(* CoDeSys 2.3.9.47 project: 3floor_2016_11_08_spalnya_fancoil_speed_temporary_change.prx *)
(* Libraries: TcEIB.lbx 16.5.14 13:12:22, TcSystemBX.lbx 11.6.12 12:56:16, TcBABasicBX.lbx 22.7.15 14:46:56, TcBaseBX.lbx 10.5.06 07:50:20, standard.lbx 5.12.03 07:02:30 *)

(* Task configuration *)
TASK Standard (PRIORITY := 0, INTERVAL := T#20ms);
	MAIN
END_TASK

(* Global variable list: M_Var_1 *)
VAR_GLOBAL
	data1floor: ARRAY[0..200] OF BYTE;
	data1floor_prev: ARRAY[0..200] OF BYTE;
	ads_adr1: STRING:='10.0.5.61.1.1';

	fb_komora_l_send_status_ex: 			EIB_BIT_SEND_EX;
	fb_su1_l_send_status_ex: 				EIB_BIT_SEND_EX;
	fb_topochna_l_send_status_ex: 			EIB_BIT_SEND_EX;
	fb_su2_bra_send_status_ex: 				EIB_BIT_SEND_EX;
	fb_topochna2_l_send_status_ex: 		EIB_BIT_SEND_EX;
	fb_su2_l_send_status_ex: 				EIB_BIT_SEND_EX;
	fb_su1_rakovyna_send_status_ex: 		EIB_BIT_SEND_EX;
	fb_su2_dush_send_status_ex: 			EIB_BIT_SEND_EX;
	fb_dush_send_status_ex: 				EIB_BIT_SEND_EX;
	fb_vitalnya_smugy2_send_status_ex: 		EIB_BIT_SEND_EX;
	fb_su2_polytsi_send_status_ex: 			EIB_BIT_SEND_EX;
	fb_kuhnya1_send_status_ex: 			EIB_BIT_SEND_EX;
	fb_kuhnya2_send_status_ex: 			EIB_BIT_SEND_EX;
	fb_vitalnya_smugy1_send_status_ex: 		EIB_BIT_SEND_EX;
	fb_vitalnya_l_send_status_ex: 			EIB_BIT_SEND_EX;
	fb_vitalnya_prokladka_send_status_ex: 	EIB_BIT_SEND_EX;
	fb_terassa_stina_send_status_ex: 		EIB_BIT_SEND_EX;
	fb_pidval_shody_send_status_ex: 		EIB_BIT_SEND_EX;
	fb_skhody2pov_send_status_ex: 			EIB_BIT_SEND_EX;
	fb_tambur_l_send_status_ex: 			EIB_BIT_SEND_EX;
	fb_vent_su1_send_status_ex: 			EIB_BIT_SEND_EX;
	fb_vent_kuh_low_send_status_ex: 		EIB_BIT_SEND_EX;
	fb_vent_dush_send_status_ex: 			EIB_BIT_SEND_EX;
	fb_vent_komora_send_status_ex: 		EIB_BIT_SEND_EX;
	fb_vent_kuh_high_send_status_ex: 		EIB_BIT_SEND_EX;
	fb_floor1_lights_send_status_ex: 			EIB_BIT_SEND_EX;

	fb_komora_l_read: 			EIB_BIT_REC;
	fb_su1_l_read: 				EIB_BIT_REC;
	fb_topochna_l_read: 		EIB_BIT_REC;
	fb_su2_bra_read: 			EIB_BIT_REC;
	fb_topochna2_l_read: 		EIB_BIT_REC;
	fb_su2_l_read: 				EIB_BIT_REC;
	fb_su1_rakovyna_read: 		EIB_BIT_REC;
	fb_su2_dush_read: 			EIB_BIT_REC;
	fb_dush_read: 				EIB_BIT_REC;
	fb_vitalnya_smugy2_read: 	EIB_BIT_REC;
	fb_su2_polytsi_read: 		EIB_BIT_REC;
	fb_kuhnya1_read: 			EIB_BIT_REC;
	fb_kuhnya2_read: 			EIB_BIT_REC;
	fb_vitalnya_smugy1_read: 	EIB_BIT_REC;
	fb_vitalnya_l_read: 			EIB_BIT_REC;
	fb_vitalnya_prokladka_read: 	EIB_BIT_REC;
	fb_terassa_stina_read: 		EIB_BIT_REC;
	fb_pidval_shody_read: 		EIB_BIT_REC;
	fb_skhody2pov_read: 		EIB_BIT_REC;
	fb_tambur_l_read: 			EIB_BIT_REC;
	fb_vent_su1_read: 			EIB_BIT_REC;
	fb_vent_kuh_low_read: 		EIB_BIT_REC;
	fb_vent_dush_read: 			EIB_BIT_REC;
	fb_vent_komora_read: 		EIB_BIT_REC;
	fb_vent_kuh_high_read: 		EIB_BIT_REC;
	fb_floor1_lights_read: 		EIB_BIT_REC;

	moove_garderob				AT%MX100.0:BOOL;
	moove_tambur					AT%MX100.1:BOOL;
	moove_dytjacha					AT%MX100.2:BOOL;
	moove_spalnya					AT%MX100.3:BOOL;
	moove_korydor					AT%MX100.4:BOOL;
	moove_skhody					AT%MX100.5:BOOL;

	komora_l 						AT%MX101.0:BOOL;
	su1_l 							AT%MX101.1:BOOL;
	topochna_l 						AT%MX101.2:BOOL;
	su2_bra	 						AT%MX101.3:BOOL;
	su2_l 							AT%MX101.4:BOOL;
	su1_rakovyna 					AT%MX101.5:BOOL;
	su2_dush 						AT%MX101.6:BOOL;
	dush 							AT%MX101.7:BOOL;

	kuhnya1	 					AT%MX102.0:BOOL;
	vitalnya_smugy1 				AT%MX102.1:BOOL;
	vitalnya_l 						AT%MX102.2:BOOL;
	vitalnya_prokladka 				AT%MX102.3:BOOL;
	terassa_stina	 				AT%MX102.4:BOOL;
	pidval_shody	 				AT%MX102.5:BOOL;
	skhody2pov 					AT%MX102.6:BOOL;
	tambur_l 						AT%MX102.7:BOOL;

	vent_su1 						AT%MX103.0:BOOL;
	vent_kuh_low 					AT%MX103.1:BOOL;
	vent_dush 						AT%MX103.2:BOOL;
	vent_komora 					AT%MX103.3:BOOL;
	vent_kuh_high 					AT%MX103.4:BOOL;

	floor1_lights:						BOOL;

END_VAR

(* Global variable list: M_Var_2 *)
VAR_GLOBAL
	data2floor: ARRAY[0..300] OF BYTE;
	data2floor_prev: ARRAY[0..300] OF BYTE;
	ads_adr2: STRING:='10.0.5.62.1.1';

	fb_balkon_peryla_send_status_ex: 			EIB_BIT_SEND_EX;
	fb_kino_l_send_status_ex:  					EIB_BIT_SEND_EX;
	fb_balkon_bra_send_status_ex: 				EIB_BIT_SEND_EX;
	fb_kabinet_balkon_l_send_status_ex:  		EIB_BIT_SEND_EX;
	fb_balkon_send_status_ex:					EIB_BIT_SEND_EX;
	fb_korydor1_send_status_ex:	 				EIB_BIT_SEND_EX;
	fb_kino_bra_send_status_ex:					EIB_BIT_SEND_EX;
	fb_kino_bra_send_dim_status_ex:			EIB_8BIT_SIGN_SEND_EX;
	fb_studio_pidsvitka_send_status_ex: 			EIB_BIT_SEND_EX;
	fb_skhody2_3_send_status_ex:	  			EIB_BIT_SEND_EX;
	fb_studio_l_send_status_ex:	 				EIB_BIT_SEND_EX;
	fb_kabinet_svitlo_send_status_ex:			EIB_BIT_SEND_EX;
	fb_stend_send_status_ex:  					EIB_BIT_SEND_EX;
	fb_kabinet_kobra_send_status_ex:  			EIB_BIT_SEND_EX;
	fb_skhody_peryla_send_status_ex:  			EIB_BIT_SEND_EX;
	fb_tambur2_send_status_ex: 					EIB_BIT_SEND_EX;
	fb_floor2_lights_send_status_ex: 				EIB_BIT_SEND_EX;

	fb_balkon_peryla_read: 						EIB_BIT_REC;
	fb_kino_l_read:  								EIB_BIT_REC;
	fb_balkon_bra_read: 						EIB_BIT_REC;
	fb_kabinet_balkon_l_read:  					EIB_BIT_REC;
	fb_balkon_read:								EIB_BIT_REC;
	fb_korydor1_read:							EIB_BIT_REC;
	fb_kino_bra_read:							EIB_BIT_REC;
	fb_kino_bra_dim_read:						EIB_8BIT_SIGN_REC;
	fb_studio_pidsvitka_read: 					EIB_BIT_REC;
	fb_skhody2_3_read:	  						EIB_BIT_REC;
	fb_studio_l_read:	 						EIB_BIT_REC;
	fb_kabinet_svitlo_read:						EIB_BIT_REC;
	fb_stend_read:  								EIB_BIT_REC;
	fb_kabinet_kobra_read:  						EIB_BIT_REC;
	fb_skhody_peryla_read:  						EIB_BIT_REC;
	fb_tambur2_read: 							EIB_BIT_REC;
	fb_floor2_lights_read: 						EIB_BIT_REC;


	eib_shtory_kino, eib_tul_kino: 				EIB_BIT_REC; (*ловлять в мережі смартбаса телеграмки для штор і тюлей*)
	eib_shtory_kabinet, eib_tul_kabinet: 			EIB_BIT_REC;

	fb_eib_shtory_kino_move:					EIB_BIT_REC;
	fb_eib_shtory_kino_position:					EIB_8BIT_SIGN_REC;
	fb_eib_shtory_kino_actualPosition:			EIB_8BIT_SIGN_SEND;

	fb_eib_tul_kino_move:						EIB_BIT_REC;
	fb_eib_tul_kino_position:						EIB_8BIT_SIGN_REC;
	fb_eib_tul_kino_actualPosition:				EIB_8BIT_SIGN_SEND;

	fb_eib_shtory_kabinet_move:					EIB_BIT_REC;
	fb_eib_shtory_kabinet_position:				EIB_8BIT_SIGN_REC;
	fb_eib_shtory_kabinet_actualPosition:			EIB_8BIT_SIGN_SEND;

	fb_eib_tul_kabinet_move:					EIB_BIT_REC;
	fb_eib_tul_kabinet_position:					EIB_8BIT_SIGN_REC;
	fb_eib_tul_kabinet_actualPosition:			EIB_8BIT_SIGN_SEND;






	balkon_peryla					AT%MX200.0:BOOL;
	kino_l							AT%MX200.1:BOOL;
	balkon_bra						AT%MX200.2:BOOL;
	kabinet_balkon_l				AT%MX200.3:BOOL;
	balkon							AT%MX200.4:BOOL;
	korydor1						AT%MX200.5:BOOL;
	kino_bra						AT%MX200.6:BOOL;
	studio_pidsvitka					AT%MX200.7:BOOL;

	skhody2_3						AT%MX201.0:BOOL;
	studio_l							AT%MX201.1:BOOL;
	kabinet_svitlo					AT%MX201.2:BOOL;
	kabinet_kobra					AT%MX201.3:BOOL;
	tambur2							AT%MX201.4:BOOL;
	stend							AT%MX201.5:BOOL;
	skhody_peryla					AT%MX201.6:BOOL;

	kino_bra_dim_value				AT%MB202:BYTE;

	collector_kabinet1					AT%MX203.0:BOOL;
	collector_kabinet2					AT%MX203.1:BOOL;
	collector_studio1					AT%MX203.2:BOOL;
	collector_studio2					AT%MX203.3:BOOL;

	fancoil_kabinet_low					AT%MX203.4:BOOL;
	fancoil_kabinet_med					AT%MX203.5:BOOL;
	fancoil_kabinet_high					AT%MX203.6:BOOL;

	fancoil_kino_low						AT%MX203.7:BOOL;
	fancoil_kino_med					AT%MX204.0:BOOL;
	fancoil_kino_high					AT%MX204.1:BOOL;


	kino_shtory_ActualPosition		AT%MB205:USINT;
	kino_tul_ActualPosition			AT%MB206:USINT;
	kabinet_shtory_ActualPosition	AT%MB207:USINT;
	kabinet_tul_ActualPosition		AT%MB208:USINT;

	kabinet_floor_T_byte0			AT%MB209:BYTE;
	kabinet_floor_T_byte1			AT%MB210:BYTE;
	kabinet_floor_T_byte2			AT%MB211:BYTE;
	kabinet_floor_T_byte3			AT%MB212:BYTE;

	studio_floor_T_byte0				AT%MB213:BYTE;
	studio_floor_T_byte1				AT%MB214:BYTE;
	studio_floor_T_byte2				AT%MB215:BYTE;
	studio_floor_T_byte3				AT%MB216:BYTE;

	floor2_lights:						BOOL;
END_VAR

(* Global variable list: M_Var_4 *)
VAR_GLOBAL

	data_derevo: ARRAY[0..300] OF BYTE;
	data_derevo_prev: ARRAY[0..300] OF BYTE;
	ads_adr4: STRING:='10.0.5.64.1.1';



	fb_derevo_vidpochynok1_send_status_ex: 		EIB_BIT_SEND_EX;
	fb_derevo_vidpochynok2_send_status_ex: 		EIB_BIT_SEND_EX;
	fb_derevo_veranda_send_status_ex: 				EIB_BIT_SEND_EX;
	fb_derevo_veranda_zovn_send_status_ex: 		EIB_BIT_SEND_EX;
	fb_derevo_vhid_zovn_send_status_ex: 			EIB_BIT_SEND_EX;
	fb_derevo_sauna_send_status_ex: 				EIB_BIT_SEND_EX;
	fb_derevo_vhid_send_status_ex: 				EIB_BIT_SEND_EX;
	fb_derevo_kotel_send_status_ex: 				EIB_BIT_SEND_EX;
	fb_derevo_korydor_send_status_ex: 				EIB_BIT_SEND_EX;
	fb_derevo_sinna_send_status_ex: 				EIB_BIT_SEND_EX;
	fb_derevo_hamam_send_status_ex: 				EIB_BIT_SEND_EX;
	fb_derevo_kuhnya_send_status_ex: 				EIB_BIT_SEND_EX;
	fb_derevo_bassein1_send_status_ex: 			EIB_BIT_SEND_EX;
	fb_derevo_bassein_lampa_send_status_ex: 		EIB_BIT_SEND_EX;
	fb_derevo_spalnya2_send_status_ex: 			EIB_BIT_SEND_EX;
	fb_derevo_terassa_send_status_ex: 				EIB_BIT_SEND_EX;
	fb_derevo_dush_send_status_ex: 				EIB_BIT_SEND_EX;
	fb_derevo_wc_send_status_ex: 					EIB_BIT_SEND_EX;
	fb_derevo_spalnya_verh_send_status_ex: 		EIB_BIT_SEND_EX;
	fb_derevo_spalnya1_send_status_ex: 			EIB_BIT_SEND_EX;
	fb_derevo_spalnya_su_send_status_ex: 			EIB_BIT_SEND_EX;
	fb_derevo_garderob_send_status_ex: 			EIB_BIT_SEND_EX;
	fb_derevo_dush2_send_status_ex: 				EIB_BIT_SEND_EX;
	fb_derevo_okno_basseina_send_status_ex: 		EIB_BIT_SEND_EX;
	fb_derevo_lights_send_status_ex: 				EIB_BIT_SEND_EX;

	fb_derevo_vidpochynok1_read: 		EIB_BIT_REC;
	fb_derevo_vidpochynok2_read: 		EIB_BIT_REC;
	fb_derevo_veranda_read: 			EIB_BIT_REC;
	fb_derevo_veranda_zovn_read: 		EIB_BIT_REC;
	fb_derevo_vhid_zovn_read: 			EIB_BIT_REC;
	fb_derevo_sauna_read: 				EIB_BIT_REC;
	fb_derevo_vhid_read: 				EIB_BIT_REC;
	fb_derevo_kotel_read: 				EIB_BIT_REC;
	fb_derevo_korydor_read:				EIB_BIT_REC;
	fb_derevo_sinna_read: 				EIB_BIT_REC;
	fb_derevo_hamam_read: 			EIB_BIT_REC;
	fb_derevo_kuhnya_read: 			EIB_BIT_REC;
	fb_derevo_bassein1_read: 			EIB_BIT_REC;
	fb_derevo_bassein_lampa_read: 		EIB_BIT_REC;
	fb_derevo_spalnya2_read: 			EIB_BIT_REC;
	fb_derevo_terassa_read: 			EIB_BIT_REC;
	fb_derevo_dush_read: 				EIB_BIT_REC;
	fb_derevo_wc_read: 				EIB_BIT_REC;
	fb_derevo_spalnya_verh_read: 		EIB_BIT_REC;
	fb_derevo_spalnya1_read: 			EIB_BIT_REC;
	fb_derevo_spalnya_su_read: 		EIB_BIT_REC;
	fb_derevo_garderob_read: 			EIB_BIT_REC;
	fb_derevo_dush2_read: 				EIB_BIT_REC;
	fb_derevo_okno_basseina_read: 		EIB_BIT_REC;
	fb_derevo_lights_read: 				EIB_BIT_REC;

	derevo_vidpochynok1 		AT %MX500.0:	 BOOL;
	derevo_vidpochynok2 		AT %MX500.1:	 BOOL;
	derevo_veranda 			AT %MX500.2:	 BOOL;
	derevo_veranda_zovn 		AT %MX500.3:	 BOOL;
	derevo_vhid_zovn 			AT %MX500.4:	 BOOL;
	derevo_sauna 				AT %MX500.5:	 BOOL;
	derevo_vhid					AT %MX500.6:	 BOOL;
	derevo_kotel 				AT %MX500.7:	 BOOL;

	derevo_korydor 				AT %MX501.0:	 BOOL;
	derevo_sinna 				AT %MX501.1:	 BOOL;
	derevo_hamam 				AT %MX501.2:	 BOOL;
	derevo_kuhnya 				AT %MX501.3:	 BOOL;
	derevo_bassein1			AT %MX501.4:	 BOOL;
	derevo_bassein_lampa		AT %MX501.5:	 BOOL;
	derevo_spalnya2			AT %MX501.6:	 BOOL;
	derevo_terassa 				AT %MX501.7:	 BOOL;

	derevo_dush 				AT %MX502.0:	 BOOL;
	derevo_wc 					AT %MX502.1:	 BOOL;
	derevo_spalnya_verh		AT %MX502.2:	 BOOL;
	derevo_spalnya1 			AT %MX502.3:	 BOOL;
	derevo_spalnya_su 			AT %MX502.4:	 BOOL;
	derevo_garderob 			AT %MX502.5:	 BOOL;
	derevo_dush2				AT %MX502.6:	 BOOL;
	derevo_okno_basseina		AT %MX503.0:	 BOOL;

	derevo_lights:						BOOL;
END_VAR

(* Global variable list: main *)
VAR_GLOBAL


	bDarkOutside: BOOL;
	t_out:REAL;
	OAT:INT;
	fb_KL6301_0: KL6301; (* EIB functonblock *)
	system_time:timestruct;

	VITALNYA_HVAC: ROOM_HVAC;
	SPALNYA_HVAC: ROOM_HVAC;
	DYTJACHA_HVAC: ROOM_HVAC;
	KINO_HVAC:ROOM_HVAC;
	STUDIO_HVAC: ROOM_HVAC;
	KABINET_HVAC:ROOM_HVAC;

	heating_mode:BOOL:=TRUE; (*false means COOLING*)

(*global parameters eib adresses*)
	heating_mode_addr:EIB_GROUP_ADDR:= (MAIN:=1, SUB_MAIN:=2, NUMBER:=10);

(*adresses for Temperatures from HDL panels *)







(*adresses for actual setpoint from eib_port *)
(*adresses for current speed and setpoint of cooling mode from HDL panels *)

(*adresses for current speed and setpoint of heating mode from HDL panels *)



	vitalnya_T_EIB_addr: 								EIB_GROUP_ADDR:= (MAIN:=1, SUB_MAIN:=1, NUMBER:=0);
	vitalnya_cooling_EIB_addr: 							EIB_GROUP_ADDR:= (MAIN:=1, SUB_MAIN:=1, NUMBER:=1);
	vitalnya_heating_EIB_addr: 							EIB_GROUP_ADDR:= (MAIN:=1, SUB_MAIN:=1, NUMBER:=2);
	vitalnya_fan_EIB_addr: 								EIB_GROUP_ADDR:= (MAIN:=1, SUB_MAIN:=1, NUMBER:=3);

	vitalnya_actual_setpoint_addr: 						EIB_GROUP_ADDR:= (MAIN:=1, SUB_MAIN:=1, NUMBER:=5);
	vitalnya_FCU_heating_ctrl_sig_EIB_addr: 				EIB_GROUP_ADDR:= (MAIN:=1, SUB_MAIN:=1, NUMBER:=6);
	vitalnya_FCU_cooling_ctrl_sig_EIB_addr: 				EIB_GROUP_ADDR:= (MAIN:=1, SUB_MAIN:=1, NUMBER:=7);
	vitalnya_FCU_fan_speed_EIB_addr:					EIB_GROUP_ADDR:= (MAIN:=1, SUB_MAIN:=1, NUMBER:=8);

	komora_l_adr: 										EIB_GROUP_ADDR:= (MAIN:=1, SUB_MAIN:=1, NUMBER:=10);
	su1_l_adr: 											EIB_GROUP_ADDR:= (MAIN:=1, SUB_MAIN:=1, NUMBER:=11);
	topochna_l_adr:	 									EIB_GROUP_ADDR:= (MAIN:=1, SUB_MAIN:=1, NUMBER:=12);
	su2_bra_adr:	 									EIB_GROUP_ADDR:= (MAIN:=1, SUB_MAIN:=1, NUMBER:=13);
	su2_l_adr:	 										EIB_GROUP_ADDR:= (MAIN:=1, SUB_MAIN:=1, NUMBER:=14);
	su1_rakovyna_adr:	 								EIB_GROUP_ADDR:= (MAIN:=1, SUB_MAIN:=1, NUMBER:=15);
	su2_dush_adr:	 									EIB_GROUP_ADDR:= (MAIN:=1, SUB_MAIN:=1, NUMBER:=16);
	dush_adr:	 										EIB_GROUP_ADDR:= (MAIN:=1, SUB_MAIN:=1, NUMBER:=17);
	kuhnya1_adr:	 									EIB_GROUP_ADDR:= (MAIN:=1, SUB_MAIN:=1, NUMBER:=18);
	vitalnya_smugy1_adr: 								EIB_GROUP_ADDR:= (MAIN:=1, SUB_MAIN:=1, NUMBER:=19);
	vitalnya_l_adr: 										EIB_GROUP_ADDR:= (MAIN:=1, SUB_MAIN:=1, NUMBER:=20);
	vitalnya_prokladka_adr: 								EIB_GROUP_ADDR:= (MAIN:=1, SUB_MAIN:=1, NUMBER:=21);
	terassa_stina_adr: 									EIB_GROUP_ADDR:= (MAIN:=1, SUB_MAIN:=1, NUMBER:=22);
	pidval_shody_adr: 									EIB_GROUP_ADDR:= (MAIN:=1, SUB_MAIN:=1, NUMBER:=23);
	skhody2pov_adr: 									EIB_GROUP_ADDR:= (MAIN:=1, SUB_MAIN:=1, NUMBER:=24);
	tambur_l_adr:										EIB_GROUP_ADDR:= (MAIN:=1, SUB_MAIN:=1, NUMBER:=25);
	vent_su1_adr: 										EIB_GROUP_ADDR:= (MAIN:=1, SUB_MAIN:=1, NUMBER:=26);
	vent_kuh_low_adr: 									EIB_GROUP_ADDR:= (MAIN:=1, SUB_MAIN:=1, NUMBER:=27);
	vent_dush_adr: 										EIB_GROUP_ADDR:= (MAIN:=1, SUB_MAIN:=1, NUMBER:=28);
	vent_komora_adr: 									EIB_GROUP_ADDR:= (MAIN:=1, SUB_MAIN:=1, NUMBER:=29);
	vent_kuh_high_adr: 									EIB_GROUP_ADDR:= (MAIN:=1, SUB_MAIN:=1, NUMBER:=30);


	komora_l_status_adr: 								EIB_GROUP_ADDR:= (MAIN:=1, SUB_MAIN:=1, NUMBER:=110);
	su1_l_status_adr: 									EIB_GROUP_ADDR:= (MAIN:=1, SUB_MAIN:=1, NUMBER:=111);
	topochna_l_status_adr:	 							EIB_GROUP_ADDR:= (MAIN:=1, SUB_MAIN:=1, NUMBER:=112);
	su2_bra_status_adr:	 								EIB_GROUP_ADDR:= (MAIN:=1, SUB_MAIN:=1, NUMBER:=113);
	su2_l_status_adr:	 								EIB_GROUP_ADDR:= (MAIN:=1, SUB_MAIN:=1, NUMBER:=114);
	su1_rakovyna_status_adr:	 						EIB_GROUP_ADDR:= (MAIN:=1, SUB_MAIN:=1, NUMBER:=115);
	su2_dush_status_adr:	 							EIB_GROUP_ADDR:= (MAIN:=1, SUB_MAIN:=1, NUMBER:=116);
	dush_status_adr:	 								EIB_GROUP_ADDR:= (MAIN:=1, SUB_MAIN:=1, NUMBER:=117);
	kuhnya1_status_adr:	 								EIB_GROUP_ADDR:= (MAIN:=1, SUB_MAIN:=1, NUMBER:=118);
	vitalnya_smugy1_status_adr: 							EIB_GROUP_ADDR:= (MAIN:=1, SUB_MAIN:=1, NUMBER:=119);
	vitalnya_l_status_adr: 								EIB_GROUP_ADDR:= (MAIN:=1, SUB_MAIN:=1, NUMBER:=120);
	vitalnya_prokladka_status_adr: 						EIB_GROUP_ADDR:= (MAIN:=1, SUB_MAIN:=1, NUMBER:=121);
	terassa_stina_status_adr: 							EIB_GROUP_ADDR:= (MAIN:=1, SUB_MAIN:=1, NUMBER:=122);
	pidval_shody_status_adr: 							EIB_GROUP_ADDR:= (MAIN:=1, SUB_MAIN:=1, NUMBER:=123);
	skhody2pov_status_adr: 								EIB_GROUP_ADDR:= (MAIN:=1, SUB_MAIN:=1, NUMBER:=124);
	tambur_l_status_adr:									EIB_GROUP_ADDR:= (MAIN:=1, SUB_MAIN:=1, NUMBER:=125);
	vent_su1_status_adr: 								EIB_GROUP_ADDR:= (MAIN:=1, SUB_MAIN:=1, NUMBER:=126);
	vent_kuh_low_status_adr: 							EIB_GROUP_ADDR:= (MAIN:=1, SUB_MAIN:=1, NUMBER:=127);
	vent_dush_status_adr: 								EIB_GROUP_ADDR:= (MAIN:=1, SUB_MAIN:=1, NUMBER:=128);
	vent_komora_status_adr: 							EIB_GROUP_ADDR:= (MAIN:=1, SUB_MAIN:=1, NUMBER:=129);
	vent_kuh_high_status_adr: 							EIB_GROUP_ADDR:= (MAIN:=1, SUB_MAIN:=1, NUMBER:=130);

	kino_T_EIB_addr: 									EIB_GROUP_ADDR:= (MAIN:=1, SUB_MAIN:=2, NUMBER:=0);
	kino_cooling_EIB_addr: 								EIB_GROUP_ADDR:= (MAIN:=1, SUB_MAIN:=2, NUMBER:=1);
	kino_heating_EIB_addr: 								EIB_GROUP_ADDR:= (MAIN:=1, SUB_MAIN:=2, NUMBER:=2);
	kino_fan_EIB_addr: 									EIB_GROUP_ADDR:= (MAIN:=1, SUB_MAIN:=2, NUMBER:=3);
	kino_actual_setpoint_addr: 							EIB_GROUP_ADDR:= (MAIN:=1, SUB_MAIN:=2, NUMBER:=5);
	kino_FCU_heating_ctrl_sig_EIB_addr: 				EIB_GROUP_ADDR:= (MAIN:=1, SUB_MAIN:=2, NUMBER:=6);
	kino_FCU_cooling_ctrl_sig_EIB_addr: 				EIB_GROUP_ADDR:= (MAIN:=1, SUB_MAIN:=2, NUMBER:=7);
	kino_FCU_fan_speed_EIB_addr: 						EIB_GROUP_ADDR:= (MAIN:=1, SUB_MAIN:=2, NUMBER:=8);


(*adresses for damper  control and indication*)
	vitalnya_damper_EIB_addr: 							EIB_GROUP_ADDR:= (MAIN:=1, SUB_MAIN:=2, NUMBER:=10);
	kino_damper_EIB_addr: 								EIB_GROUP_ADDR:= (MAIN:=1, SUB_MAIN:=2, NUMBER:=11);
	kabinet_damper_EIB_addr: 							EIB_GROUP_ADDR:= (MAIN:=1, SUB_MAIN:=2, NUMBER:=12);
	dytjacha_damper_EIB_addr: 							EIB_GROUP_ADDR:= (MAIN:=1, SUB_MAIN:=2, NUMBER:=13);
	spalnya_damper_EIB_addr: 							EIB_GROUP_ADDR:= (MAIN:=1, SUB_MAIN:=2, NUMBER:=14);

(**adresses for shtory*)
	move_shtory_kino_EIB_addr: 						EIB_GROUP_ADDR := (MAIN:=1, SUB_MAIN:=2, NUMBER:=20);
	position_shtory_kino_EIB_addr: 						EIB_GROUP_ADDR := (MAIN:=1, SUB_MAIN:=2, NUMBER:=21);
	actrualPosition_shtory_kino_EIB_addr: 				EIB_GROUP_ADDR := (MAIN:=1, SUB_MAIN:=2, NUMBER:=22);

	move_tul_kino_EIB_addr: 							EIB_GROUP_ADDR := (MAIN:=1, SUB_MAIN:=2, NUMBER:=23);
	position_tul_kino_EIB_addr: 							EIB_GROUP_ADDR := (MAIN:=1, SUB_MAIN:=2, NUMBER:=24);
	actrualPosition_tul_kino_EIB_addr: 					EIB_GROUP_ADDR := (MAIN:=1, SUB_MAIN:=2, NUMBER:=25);

	move_shtory_kabinet_EIB_addr: 						EIB_GROUP_ADDR := (MAIN:=1, SUB_MAIN:=2, NUMBER:=26);
	position_shtory_kabinet_EIB_addr: 					EIB_GROUP_ADDR := (MAIN:=1, SUB_MAIN:=2, NUMBER:=27);
	actrualPosition_shtory_kabinet_EIB_addr: 			EIB_GROUP_ADDR := (MAIN:=1, SUB_MAIN:=2, NUMBER:=28);

	move_tul_kabinet_EIB_addr: 						EIB_GROUP_ADDR := (MAIN:=1, SUB_MAIN:=2, NUMBER:=29);
	position_tul_kabinet_EIB_addr: 						EIB_GROUP_ADDR := (MAIN:=1, SUB_MAIN:=2, NUMBER:=30);
	actrualPosition_tul_kabinet_EIB_addr: 				EIB_GROUP_ADDR := (MAIN:=1, SUB_MAIN:=2, NUMBER:=31);

(*eib date and time adresses*)
	studio_T_EIB_addr: 									EIB_GROUP_ADDR:= (MAIN:=1, SUB_MAIN:=3, NUMBER:=0);
	studio_cooling_EIB_addr: 							EIB_GROUP_ADDR:= (MAIN:=1, SUB_MAIN:=3, NUMBER:=1);
	studio_heating_EIB_addr: 							EIB_GROUP_ADDR:= (MAIN:=1, SUB_MAIN:=3, NUMBER:=2);
	studio_fan_EIB_addr: 								EIB_GROUP_ADDR:= (MAIN:=1, SUB_MAIN:=3, NUMBER:=3);
	studio_actual_setpoint_addr: 							EIB_GROUP_ADDR:= (MAIN:=1, SUB_MAIN:=3, NUMBER:=5);
	studio_FCU_fan_speed_EIB_addr: 					EIB_GROUP_ADDR:= (MAIN:=1, SUB_MAIN:=3, NUMBER:=8);
	eib_time_EIB_addr:									EIB_GROUP_ADDR :=(MAIN:=1, SUB_MAIN:=3, NUMBER:=10);
	eib_date_EIB_addr:									EIB_GROUP_ADDR :=(MAIN:=1, SUB_MAIN:=3, NUMBER:=11);
	eib_twillight_EIB_addr:								EIB_GROUP_ADDR :=(MAIN:=1, SUB_MAIN:=3, NUMBER:=12);

	kabinet_T_EIB_addr: 								EIB_GROUP_ADDR:= (MAIN:=1, SUB_MAIN:=4, NUMBER:=0);
	kabinet_cooling_EIB_addr: 							EIB_GROUP_ADDR:= (MAIN:=1, SUB_MAIN:=4, NUMBER:=1);
	kabinet_heating_EIB_addr: 							EIB_GROUP_ADDR:= (MAIN:=1, SUB_MAIN:=4, NUMBER:=2);
	kabinet_fan_EIB_addr: 								EIB_GROUP_ADDR:= (MAIN:=1, SUB_MAIN:=4, NUMBER:=3);
	kabinet_actual_setpoint_addr: 						EIB_GROUP_ADDR:= (MAIN:=1, SUB_MAIN:=4, NUMBER:=5);
	kabinet_FCU_heating_ctrl_sig_EIB_addr: 				EIB_GROUP_ADDR:= (MAIN:=1, SUB_MAIN:=4, NUMBER:=6);
	kabinet_FCU_cooling_ctrl_sig_EIB_addr: 				EIB_GROUP_ADDR:= (MAIN:=1, SUB_MAIN:=4, NUMBER:=7);
	kabinet_FCU_fan_speed_EIB_addr: 					EIB_GROUP_ADDR:= (MAIN:=1, SUB_MAIN:=4, NUMBER:=8);

	balkon_peryla_adr: 									EIB_GROUP_ADDR:= (MAIN:=1, SUB_MAIN:=4, NUMBER:=9);
	kino_l_adr: 											EIB_GROUP_ADDR:= (MAIN:=1, SUB_MAIN:=4, NUMBER:=10);
	balkon_bra_adr:	 									EIB_GROUP_ADDR:= (MAIN:=1, SUB_MAIN:=4, NUMBER:=11);
	kabinet_balkon_l_adr:	 							EIB_GROUP_ADDR:= (MAIN:=1, SUB_MAIN:=4, NUMBER:=12);
	balkon_adr:	 										EIB_GROUP_ADDR:= (MAIN:=1, SUB_MAIN:=4, NUMBER:=13);
	korydor1_adr:	 									EIB_GROUP_ADDR:= (MAIN:=1, SUB_MAIN:=4, NUMBER:=14);
	kino_bra_adr:	 									EIB_GROUP_ADDR:= (MAIN:=1, SUB_MAIN:=4, NUMBER:=15);
	kino_bra_dimming_adr:								EIB_GROUP_ADDR:= (MAIN:=1, SUB_MAIN:=4, NUMBER:=16);
	studio_pidsvitka_adr:	 							EIB_GROUP_ADDR:= (MAIN:=1, SUB_MAIN:=4, NUMBER:=17);
	skhody2_3_adr:	 									EIB_GROUP_ADDR:= (MAIN:=1, SUB_MAIN:=4, NUMBER:=18);
	studio_l_adr:	 									EIB_GROUP_ADDR:= (MAIN:=1, SUB_MAIN:=4, NUMBER:=19);
	kabinet_svitlo_adr:		 							EIB_GROUP_ADDR:= (MAIN:=1, SUB_MAIN:=4, NUMBER:=20);
	stend_adr:	 										EIB_GROUP_ADDR:= (MAIN:=1, SUB_MAIN:=4, NUMBER:=21);
	kabinet_kobra_adr:	 								EIB_GROUP_ADDR:= (MAIN:=1, SUB_MAIN:=4, NUMBER:=22);
	skhody_peryla_adr:	 								EIB_GROUP_ADDR:= (MAIN:=1, SUB_MAIN:=4, NUMBER:=23);
	tambur2_adr:	 									EIB_GROUP_ADDR:= (MAIN:=1, SUB_MAIN:=4, NUMBER:=24);

	balkon_peryla_status_adr: 							EIB_GROUP_ADDR:= (MAIN:=1, SUB_MAIN:=4, NUMBER:=109);
	kino_l_status_adr: 									EIB_GROUP_ADDR:= (MAIN:=1, SUB_MAIN:=4, NUMBER:=110);
	balkon_bra_status_adr:	 							EIB_GROUP_ADDR:= (MAIN:=1, SUB_MAIN:=4, NUMBER:=111);
	kabinet_balkon_l_status_adr:	 						EIB_GROUP_ADDR:= (MAIN:=1, SUB_MAIN:=4, NUMBER:=112);
	balkon_status_adr:	 								EIB_GROUP_ADDR:= (MAIN:=1, SUB_MAIN:=4, NUMBER:=113);
	korydor1_status_adr:	 								EIB_GROUP_ADDR:= (MAIN:=1, SUB_MAIN:=4, NUMBER:=114);
	kino_bra_status_adr:	 								EIB_GROUP_ADDR:= (MAIN:=1, SUB_MAIN:=4, NUMBER:=115);
	studio_pidsvitka_status_adr:	 						EIB_GROUP_ADDR:= (MAIN:=1, SUB_MAIN:=4, NUMBER:=117);
	skhody2_3_status_adr:	 							EIB_GROUP_ADDR:= (MAIN:=1, SUB_MAIN:=4, NUMBER:=118);
	studio_l_status_adr:	 								EIB_GROUP_ADDR:= (MAIN:=1, SUB_MAIN:=4, NUMBER:=119);
	kabinet_svitlo_status_adr:		 					EIB_GROUP_ADDR:= (MAIN:=1, SUB_MAIN:=4, NUMBER:=120);
	stend_status_adr:	 								EIB_GROUP_ADDR:= (MAIN:=1, SUB_MAIN:=4, NUMBER:=121);
	kabinet_kobra_status_adr:	 						EIB_GROUP_ADDR:= (MAIN:=1, SUB_MAIN:=4, NUMBER:=122);
	skhody_peryla_status_adr:	 						EIB_GROUP_ADDR:= (MAIN:=1, SUB_MAIN:=4, NUMBER:=123);
	tambur2_status_adr:	 								EIB_GROUP_ADDR:= (MAIN:=1, SUB_MAIN:=4, NUMBER:=124);

	dytjacha_T_EIB_addr: 								EIB_GROUP_ADDR:= (MAIN:=1, SUB_MAIN:=5, NUMBER:=0);
	dytjacha_cooling_EIB_addr: 							EIB_GROUP_ADDR:= (MAIN:=1, SUB_MAIN:=5, NUMBER:=1);
	dytjacha_heating_EIB_addr: 							EIB_GROUP_ADDR:= (MAIN:=1, SUB_MAIN:=5, NUMBER:=2);
	dytjacha_fan_EIB_addr: 								EIB_GROUP_ADDR:= (MAIN:=1, SUB_MAIN:=5, NUMBER:=3);
	dytjacha_actual_setpoint_addr: 						EIB_GROUP_ADDR:= (MAIN:=1, SUB_MAIN:=5, NUMBER:=5);
	dytjacha_FCU_heating_ctrl_sig_EIB_addr: 			EIB_GROUP_ADDR:= (MAIN:=1, SUB_MAIN:=5, NUMBER:=6);
	dytjacha_FCU_cooling_ctrl_sig_EIB_addr: 			EIB_GROUP_ADDR:= (MAIN:=1, SUB_MAIN:=5, NUMBER:=7);
	dytjacha_FCU_fan_speed_EIB_addr: 					EIB_GROUP_ADDR:= (MAIN:=1, SUB_MAIN:=5, NUMBER:=8);

	move_lift_spalnya_EIB_addr: 						EIB_GROUP_ADDR := (MAIN:=1, SUB_MAIN:=5, NUMBER:=24);
	lift_spalnya_status_EIB_addr: 						EIB_GROUP_ADDR := (MAIN:=1, SUB_MAIN:=5, NUMBER:=25);

	move_shtory_spalnya_EIB_addr: 						EIB_GROUP_ADDR := (MAIN:=1, SUB_MAIN:=5, NUMBER:=26);
	position_shtory_spalnya_EIB_addr: 					EIB_GROUP_ADDR := (MAIN:=1, SUB_MAIN:=5, NUMBER:=27);
	actrualPosition_shtory_spalnya_EIB_addr: 			EIB_GROUP_ADDR := (MAIN:=1, SUB_MAIN:=5, NUMBER:=28);

	move_tul_spanya_EIB_addr: 							EIB_GROUP_ADDR := (MAIN:=1, SUB_MAIN:=5, NUMBER:=29);
	position_tul_spalnya_EIB_addr: 						EIB_GROUP_ADDR := (MAIN:=1, SUB_MAIN:=5, NUMBER:=30);
	actrualPosition_tul_spalnya_EIB_addr: 				EIB_GROUP_ADDR := (MAIN:=1, SUB_MAIN:=5, NUMBER:=31);

	lights_out_all_eib_addr:								EIB_GROUP_ADDR := (MAIN:=1, SUB_MAIN:=5, NUMBER:=10);
	lights_out_floor1_eib_addr:							EIB_GROUP_ADDR := (MAIN:=1, SUB_MAIN:=5, NUMBER:=11);
	lights_out_floor2_eib_addr:							EIB_GROUP_ADDR := (MAIN:=1, SUB_MAIN:=5, NUMBER:=12);
	lights_out_floor3_eib_addr:							EIB_GROUP_ADDR := (MAIN:=1, SUB_MAIN:=5, NUMBER:=13);
	lights_out_derevo_eib_addr:							EIB_GROUP_ADDR := (MAIN:=1, SUB_MAIN:=5, NUMBER:=14);
	lights_out_main_house_eib_addr:						EIB_GROUP_ADDR := (MAIN:=1, SUB_MAIN:=5, NUMBER:=15);



	spalnya_T_EIB_addr: 								EIB_GROUP_ADDR:= (MAIN:=1, SUB_MAIN:=6, NUMBER:=0);
	spalnya_cooling_EIB_addr: 							EIB_GROUP_ADDR:= (MAIN:=1, SUB_MAIN:=6, NUMBER:=1);
	spalnya_heating_EIB_addr: 							EIB_GROUP_ADDR:= (MAIN:=1, SUB_MAIN:=6, NUMBER:=2);
	spalnya_fan_EIB_addr: 								EIB_GROUP_ADDR:= (MAIN:=1, SUB_MAIN:=6, NUMBER:=3);
	spalnya_actual_setpoint_addr: 						EIB_GROUP_ADDR:= (MAIN:=1, SUB_MAIN:=6, NUMBER:=5);
	spalnya_FCU_heating_ctrl_sig_EIB_addr: 				EIB_GROUP_ADDR:= (MAIN:=1, SUB_MAIN:=6, NUMBER:=6);
	spalnya_FCU_cooling_ctrl_sig_EIB_addr: 				EIB_GROUP_ADDR:= (MAIN:=1, SUB_MAIN:=6, NUMBER:=7);
	spalnya_FCU_fan_speed_EIB_addr: 					EIB_GROUP_ADDR:= (MAIN:=1, SUB_MAIN:=6, NUMBER:=8);

(*adresses for light groups*)
	spalnya_kontrazhury_adr: 							EIB_GROUP_ADDR:=(MAIN:=1, SUB_MAIN:=6, NUMBER:=9);
	spalnya_balkon_adr: 								EIB_GROUP_ADDR:=(MAIN:=1, SUB_MAIN:=6, NUMBER:=10);
	spalnya_kulbaba_adr: 								EIB_GROUP_ADDR:=(MAIN:=1, SUB_MAIN:=6, NUMBER:=11);
	su3_stina_adr: 										EIB_GROUP_ADDR:=(MAIN:=1, SUB_MAIN:=6, NUMBER:=14);
	su3_pidsvitka_adr: 									EIB_GROUP_ADDR:=(MAIN:=1, SUB_MAIN:=6, NUMBER:=15);
	su3_bra_adr: 										EIB_GROUP_ADDR:=(MAIN:=1, SUB_MAIN:=6, NUMBER:=16);
	su3_kontrazhury_adr: 								EIB_GROUP_ADDR:=(MAIN:=1, SUB_MAIN:=6, NUMBER:=17);
	dytjacha_adr: 										EIB_GROUP_ADDR:=(MAIN:=1, SUB_MAIN:=6, NUMBER:=18);
	su3_vent_adr: 										EIB_GROUP_ADDR:=(MAIN:=1, SUB_MAIN:=6, NUMBER:=19);
	su3_lampa_adr: 										EIB_GROUP_ADDR:=(MAIN:=1, SUB_MAIN:=6, NUMBER:=21);
	dytjacha_bra_adr: 									EIB_GROUP_ADDR:=(MAIN:=1, SUB_MAIN:=6, NUMBER:=20);
	garderob_adr: 										EIB_GROUP_ADDR:=(MAIN:=1, SUB_MAIN:=6, NUMBER:=22);
	bar_adr: 											EIB_GROUP_ADDR:=(MAIN:=1, SUB_MAIN:=6, NUMBER:=23);
	korydor_skeli_adr: 									EIB_GROUP_ADDR:=(MAIN:=1, SUB_MAIN:=6, NUMBER:=24);
	choven_adr: 										EIB_GROUP_ADDR:=(MAIN:=1, SUB_MAIN:=6, NUMBER:=25);
	korydor_svitlo_adr: 									EIB_GROUP_ADDR:=(MAIN:=1, SUB_MAIN:=6, NUMBER:=26);
	korydor_lampa_adr: 									EIB_GROUP_ADDR:=(MAIN:=1, SUB_MAIN:=6, NUMBER:=27);
	serverna_adr: 										EIB_GROUP_ADDR:=(MAIN:=1, SUB_MAIN:=6, NUMBER:=28);
(*adresses for back compatibility*)
	DLP_lift_spalnya_EIB_addr: 							EIB_GROUP_ADDR:=(MAIN:=1, SUB_MAIN:=6, NUMBER:=29);
	DLP_tul_spalnya_EIB_addr: 							EIB_GROUP_ADDR:=(MAIN:=1, SUB_MAIN:=6, NUMBER:=30);
	DLP_shtory_spalnya_EIB_addr: 						EIB_GROUP_ADDR:=(MAIN:=1, SUB_MAIN:=6, NUMBER:=31);



	spalnya_kontrazhury_status_adr: 						EIB_GROUP_ADDR:=(MAIN:=1, SUB_MAIN:=6, NUMBER:=109);
	spalnya_balkon_status_adr: 							EIB_GROUP_ADDR:=(MAIN:=1, SUB_MAIN:=6, NUMBER:=110);
	spalnya_kulbaba_status_adr: 						EIB_GROUP_ADDR:=(MAIN:=1, SUB_MAIN:=6, NUMBER:=111);

	su3_stina_status_adr: 								EIB_GROUP_ADDR:=(MAIN:=1, SUB_MAIN:=6, NUMBER:=114);
	su3_pidsvitka_status_adr: 							EIB_GROUP_ADDR:=(MAIN:=1, SUB_MAIN:=6, NUMBER:=115);
	su3_bra_status_adr: 									EIB_GROUP_ADDR:=(MAIN:=1, SUB_MAIN:=6, NUMBER:=116);
	su3_kontrazhury_status_adr: 							EIB_GROUP_ADDR:=(MAIN:=1, SUB_MAIN:=6, NUMBER:=117);
	su3_vent_status_adr: 								EIB_GROUP_ADDR:=(MAIN:=1, SUB_MAIN:=6, NUMBER:=119);
	su3_lampa_status_adr: 								EIB_GROUP_ADDR:=(MAIN:=1, SUB_MAIN:=6, NUMBER:=121);

	dytjacha_status_adr: 								EIB_GROUP_ADDR:=(MAIN:=1, SUB_MAIN:=6, NUMBER:=118);
	dytjacha_bra_status_adr: 							EIB_GROUP_ADDR:=(MAIN:=1, SUB_MAIN:=6, NUMBER:=120);

	garderob_status_adr: 								EIB_GROUP_ADDR:=(MAIN:=1, SUB_MAIN:=6, NUMBER:=122);
	bar_status_adr: 										EIB_GROUP_ADDR:=(MAIN:=1, SUB_MAIN:=6, NUMBER:=123);
	korydor_skeli_status_adr: 							EIB_GROUP_ADDR:=(MAIN:=1, SUB_MAIN:=6, NUMBER:=124);
	choven_status_adr: 									EIB_GROUP_ADDR:=(MAIN:=1, SUB_MAIN:=6, NUMBER:=125);
	korydor_svitlo_status_adr: 							EIB_GROUP_ADDR:=(MAIN:=1, SUB_MAIN:=6, NUMBER:=126);
	korydor_lampa_status_adr: 							EIB_GROUP_ADDR:=(MAIN:=1, SUB_MAIN:=6, NUMBER:=127);
	serverna_status_adr: 								EIB_GROUP_ADDR:=(MAIN:=1, SUB_MAIN:=6, NUMBER:=128);

	out_t_EIB_addr:										EIB_GROUP_ADDR:=(MAIN:=1, SUB_MAIN:=7, NUMBER:=0);

	derevo_vidpochynok2_adr:	 						EIB_GROUP_ADDR:= (MAIN:=1, SUB_MAIN:=7, NUMBER:=1);
	derevo_veranda_adr:	 							EIB_GROUP_ADDR:= (MAIN:=1, SUB_MAIN:=7, NUMBER:=2);
	derevo_veranda_zovn_adr:	 						EIB_GROUP_ADDR:= (MAIN:=1, SUB_MAIN:=7, NUMBER:=3);
	derevo_vhid_zovn_adr:	 							EIB_GROUP_ADDR:= (MAIN:=1, SUB_MAIN:=7, NUMBER:=4);
	derevo_sauna_adr:	 								EIB_GROUP_ADDR:= (MAIN:=1, SUB_MAIN:=7, NUMBER:=5);
	derevo_vhid_adr:									EIB_GROUP_ADDR:= (MAIN:=1, SUB_MAIN:=7, NUMBER:=6);
	derevo_kotel_adr:		 							EIB_GROUP_ADDR:= (MAIN:=1, SUB_MAIN:=7, NUMBER:=7);
	derevo_korydor_adr:		 							EIB_GROUP_ADDR:= (MAIN:=1, SUB_MAIN:=7, NUMBER:=8);
	derevo_sinna_adr:		 							EIB_GROUP_ADDR:= (MAIN:=1, SUB_MAIN:=7, NUMBER:=9);
	derevo_hamam_adr:		 							EIB_GROUP_ADDR:= (MAIN:=1, SUB_MAIN:=7, NUMBER:=10);
	derevo_kuhnya_adr:	 								EIB_GROUP_ADDR:= (MAIN:=1, SUB_MAIN:=7, NUMBER:=11);
	derevo_bassein1_adr:								EIB_GROUP_ADDR:= (MAIN:=1, SUB_MAIN:=7, NUMBER:=12);
	derevo_bassein_lampa_adr:							EIB_GROUP_ADDR:= (MAIN:=1, SUB_MAIN:=7, NUMBER:=13);
	derevo_spalnya2_adr:								EIB_GROUP_ADDR:= (MAIN:=1, SUB_MAIN:=7, NUMBER:=14);
	derevo_terassa_adr:									EIB_GROUP_ADDR:= (MAIN:=1, SUB_MAIN:=7, NUMBER:=15);
	derevo_dush_adr:	 								EIB_GROUP_ADDR:= (MAIN:=1, SUB_MAIN:=7, NUMBER:=16);
	derevo_wc_adr:										EIB_GROUP_ADDR:= (MAIN:=1, SUB_MAIN:=7, NUMBER:=17);
	derevo_spalnya_verh_adr:							EIB_GROUP_ADDR:= (MAIN:=1, SUB_MAIN:=7, NUMBER:=18);
	derevo_spalnya1_adr:								EIB_GROUP_ADDR:= (MAIN:=1, SUB_MAIN:=7, NUMBER:=19);
	derevo_spalnya_su_adr:								EIB_GROUP_ADDR:= (MAIN:=1, SUB_MAIN:=7, NUMBER:=20);
	derevo_garderob_adr:								EIB_GROUP_ADDR:= (MAIN:=1, SUB_MAIN:=7, NUMBER:=21);
	derevo_vidpochynok1_adr:	 						EIB_GROUP_ADDR:= (MAIN:=1, SUB_MAIN:=7, NUMBER:=22);
	derevo_dush2_adr:									EIB_GROUP_ADDR:= (MAIN:=1, SUB_MAIN:=7, NUMBER:=23);
	derevo_okno_basseina_adr:							EIB_GROUP_ADDR:= (MAIN:=1, SUB_MAIN:=7, NUMBER:=24);

	derevo_vidpochynok2_status_adr:	 				EIB_GROUP_ADDR:= (MAIN:=1, SUB_MAIN:=7, NUMBER:=101);
	derevo_veranda_status_adr:	 						EIB_GROUP_ADDR:= (MAIN:=1, SUB_MAIN:=7, NUMBER:=102);
	derevo_veranda_zovn_status_adr:	 				EIB_GROUP_ADDR:= (MAIN:=1, SUB_MAIN:=7, NUMBER:=103);
	derevo_vhid_zovn_status_adr:	 					EIB_GROUP_ADDR:= (MAIN:=1, SUB_MAIN:=7, NUMBER:=104);
	derevo_sauna_status_adr:	 						EIB_GROUP_ADDR:= (MAIN:=1, SUB_MAIN:=7, NUMBER:=105);
	derevo_vhid_status_adr:								EIB_GROUP_ADDR:= (MAIN:=1, SUB_MAIN:=7, NUMBER:=106);
	derevo_kotel_status_adr:		 					EIB_GROUP_ADDR:= (MAIN:=1, SUB_MAIN:=7, NUMBER:=107);
	derevo_korydor_status_adr:		 					EIB_GROUP_ADDR:= (MAIN:=1, SUB_MAIN:=7, NUMBER:=108);
	derevo_sinna_status_adr:		 					EIB_GROUP_ADDR:= (MAIN:=1, SUB_MAIN:=7, NUMBER:=109);
	derevo_hamam_status_adr:		 					EIB_GROUP_ADDR:= (MAIN:=1, SUB_MAIN:=7, NUMBER:=110);
	derevo_kuhnya_status_adr:	 						EIB_GROUP_ADDR:= (MAIN:=1, SUB_MAIN:=7, NUMBER:=111);
	derevo_bassein1_status_adr:							EIB_GROUP_ADDR:= (MAIN:=1, SUB_MAIN:=7, NUMBER:=112);
	derevo_bassein_lampa_status_adr:					EIB_GROUP_ADDR:= (MAIN:=1, SUB_MAIN:=7, NUMBER:=113);
	derevo_spalnya2_status_adr:							EIB_GROUP_ADDR:= (MAIN:=1, SUB_MAIN:=7, NUMBER:=114);
	derevo_terassa_status_adr:							EIB_GROUP_ADDR:= (MAIN:=1, SUB_MAIN:=7, NUMBER:=115);
	derevo_dush_status_adr:	 						EIB_GROUP_ADDR:= (MAIN:=1, SUB_MAIN:=7, NUMBER:=116);
	derevo_wc_status_adr:								EIB_GROUP_ADDR:= (MAIN:=1, SUB_MAIN:=7, NUMBER:=117);
	derevo_spalnya_verh_status_adr:					EIB_GROUP_ADDR:= (MAIN:=1, SUB_MAIN:=7, NUMBER:=118);
	derevo_spalnya1_status_adr:							EIB_GROUP_ADDR:= (MAIN:=1, SUB_MAIN:=7, NUMBER:=119);
	derevo_spalnya_su_status_adr:						EIB_GROUP_ADDR:= (MAIN:=1, SUB_MAIN:=7, NUMBER:=120);
	derevo_garderob_status_adr:							EIB_GROUP_ADDR:= (MAIN:=1, SUB_MAIN:=7, NUMBER:=121);
	derevo_vidpochynok1_status_adr:	 				EIB_GROUP_ADDR:= (MAIN:=1, SUB_MAIN:=7, NUMBER:=122);
	derevo_dush2_status_adr:							EIB_GROUP_ADDR:= (MAIN:=1, SUB_MAIN:=7, NUMBER:=123);
	derevo_okno_basseina_status_adr:					EIB_GROUP_ADDR:= (MAIN:=1, SUB_MAIN:=7, NUMBER:=124);



	fb_spalnya_kontrazhury_send_status_ex: 			EIB_BIT_SEND_EX;
	fb_spalnya_balkon_send_status_ex: 				EIB_BIT_SEND_EX;
	fb_spalnya_kulbaba_send_status_ex: 			EIB_BIT_SEND_EX;


	fb_su3_stina_send_status_ex: 					EIB_BIT_SEND_EX;
	fb_su3_pidsvitka_send_status_ex: 				EIB_BIT_SEND_EX;
	fb_su3_bra_send_status_ex: 						EIB_BIT_SEND_EX;
	fb_su3_kontrazhur_send_status_ex: 				EIB_BIT_SEND_EX;
	fb_su3_vent_send_status_ex: 					EIB_BIT_SEND_EX;
	fb_su3_lampa_send_status_ex: 					EIB_BIT_SEND_EX;

	fb_dytjacha_send_status_ex: 					EIB_BIT_SEND_EX;
	fb_dytjacha_bra_send_status_ex: 				EIB_BIT_SEND_EX;

	fb_garderob_send_status_ex: 					EIB_BIT_SEND_EX;
	fb_bar_send_status_ex: 							EIB_BIT_SEND_EX;
	fb_korydor_skeli_send_status_ex: 				EIB_BIT_SEND_EX;
	fb_choven_send_status_ex: 						EIB_BIT_SEND_EX;
	fb_korydor_svitlo_send_status_ex: 				EIB_BIT_SEND_EX;
	fb_korydor_lampa_send_status_ex: 				EIB_BIT_SEND_EX;
	fb_serverna_send_status_ex: 					EIB_BIT_SEND_EX;
	fb_lift_send_status_ex: 							EIB_BIT_SEND_EX;
	fb_floor3_lights_send_status_ex: 					EIB_BIT_SEND_EX;
	fb_main_house_lights_send_status_ex: 			EIB_BIT_SEND_EX;
	fb_all_lights_send_status_ex: 					EIB_BIT_SEND_EX;

	fb_spalnya_kontrazhury_read: 		EIB_BIT_REC;
	fb_spalnya_balkon_read: 			EIB_BIT_REC;
	fb_spalnya_kulbaba_read: 			EIB_BIT_REC;

	fb_su3_stina_read: 					EIB_BIT_REC;
	fb_su3_pidsvitka_read: 				EIB_BIT_REC;
	fb_su3_bra_read: 					EIB_BIT_REC;
	fb_su3_kontrazhur_read: 			EIB_BIT_REC;
	fb_su3_vent_read: 					EIB_BIT_REC;
	fb_su3_lampa_read: 					EIB_BIT_REC;

	fb_dytjacha_read: 					EIB_BIT_REC;
	fb_dytjacha_bra_read: 				EIB_BIT_REC;

	fb_garderob_read: 					EIB_BIT_REC;
	fb_bar_read: 						EIB_BIT_REC;
	fb_korydor_skeli_read: 				EIB_BIT_REC;
	fb_choven_read: 					EIB_BIT_REC;
	fb_korydor_svitlo_read: 				EIB_BIT_REC;
	fb_korydor_lampa_read: 				EIB_BIT_REC;
	fb_serverna_read: 					EIB_BIT_REC;

	fb_floor3_lights_read: 				EIB_BIT_REC;
	fb_main_house_lights_read: 			EIB_BIT_REC;
	fb_all_lights_read: 					EIB_BIT_REC;


	fb_eib_shtory_spalnya_move:				EIB_BIT_REC;
	fb_eib_shtory_spalnya_position:				EIB_8BIT_SIGN_REC;
	fb_eib_shtory_spalnya_actualPosition:		EIB_8BIT_SIGN_SEND;

	fb_eib_tul_spalnya_move:					EIB_BIT_REC;
	fb_eib_tul_spalnya_position:					EIB_8BIT_SIGN_REC;
	fb_eib_tul_spalnya_actualPosition:			EIB_8BIT_SIGN_SEND;

	fb_eib_lift_spalnya_move:					EIB_BIT_REC;


	eib_spalnya_kontrazhury: 			BOOL;
	eib_spalnya_balkon: 				BOOL;
	eib_spalnya_kulbaba: 				BOOL;
	eib_su3_stina: 						BOOL;
	eib_su3_pidsvitka: 					BOOL;
	eib_su3_bra: 						BOOL;
	eib_su3_kontrazhury: 				BOOL;
	eib_su3_vent:						BOOL;
	eib_su3_lampa: 						BOOL;
	eib_dytjacha: 						BOOL;
	eib_dytjacha_bra: 					BOOL;
	eib_garderob: 						BOOL;
	eib_bar: 							BOOL;
	eib_korydor_skeli: 					BOOL;
	eib_choven: 						BOOL;
	eib_korydor_lampa: 					BOOL;
	eib_serverna: 						BOOL;
	eib_korydor_svitlo: 					BOOL;
	eib_shtory_spalnya_move:				BOOL;
	eib_shtory_spalnya_position:				USINT;
	eib_shtory_spalnya_actualPosition:		INT;

	eib_tul_spalnya_move:					BOOL;
	eib_tul_spalnya_position:					USINT;
	eib_tul_spalnya_actualPosition:			INT;
	eib_lift_spalnya_move:				BOOL;

	floor3_lights:						BOOL;
	main_house_lights:				BOOL;
	all_lights:						BOOL;

(*видалити пысля того, як перероблю штори на функцыональних блоках*)
	tLongPress: TIME;
	tOffDelay: TIME;


	ads_adr3: STRING;


	moove_sensors:BOOL;



END_VAR

(* Global variable list: physical *)
VAR_GLOBAL
	din1_1	AT %IX0.0:	BOOL;
	din1_2	AT %IX0.1:	BOOL;
	din1_3	AT %IX0.2:	BOOL;
	din1_4	AT %IX0.3:	BOOL;
	din1_5	AT %IX0.4:	BOOL;
	din1_6	AT %IX0.5:	BOOL;
	din1_7	AT %IX0.6:	BOOL;
	din1_8	AT %IX0.7:	BOOL;
	din2_1	AT %IX1.0:	BOOL;
	din2_2	AT %IX1.1:	BOOL;
	din2_3	AT %IX1.2:	BOOL;
	din2_4	AT %IX1.3:	BOOL;
	din2_5	AT %IX1.4:	BOOL;
	din2_6	AT %IX1.5:	BOOL;
	din2_7	AT %IX1.6:	BOOL;
	din2_8	AT %IX1.7:	BOOL;
	sw_garderob1	AT %IX2.0:	BOOL;
	sw_dytjacha1 	AT %IX2.1:	BOOL;
	sw_garderob2	AT %IX2.2:	BOOL;
	sw_dytjacha2		AT %IX2.3:	BOOL;
	sw_tambur3_2	AT %IX2.4:	BOOL;
	sw_korydor		AT %IX2.5:	BOOL;
	sw_tambur3_1		AT %IX2.6:	BOOL;
	din3_8			AT %IX2.7:	BOOL;
	sw_su2			AT %IX3.0:	BOOL;
	sw_spalnya3		AT %IX3.1:	BOOL;
	sw_su1			AT %IX3.2:	BOOL;
	sw_spalnya1		AT %IX3.3:	BOOL;
	sw_spalnya_balk	AT %IX3.4:	BOOL;
	sw_spalnya2		AT %IX3.5:	BOOL;
	sw_tambur2			AT %IX3.6:	BOOL;
	sw_spalnya4		AT %IX3.7:	BOOL;
(*dout1_1*)z_vitalnya	AT %QX0.0:	BOOL;
(*dout1_2*)z_spalnya	AT %QX0.1:	BOOL;
(*dout1_3*)z_kabinet	AT %QX0.2:	BOOL;
	dout1_4	AT %QX0.3:	BOOL;
(*dout1_5*)z_kino	AT %QX0.4:	BOOL;
	dout1_6	AT %QX0.5:	BOOL;
(*dout1_7*)z_dytjacha	AT %QX0.6:	BOOL;
	dout1_8	AT %QX0.7:	BOOL;
	dout2_1	AT %QX1.0:	BOOL;
	dout2_2	AT %QX1.1:	BOOL;
	dout2_3	AT %QX1.2:	BOOL;
	dout2_4	AT %QX1.3:	BOOL;
	dout2_5	AT %QX1.4:	BOOL;
	dout2_6	AT %QX1.5:	BOOL;
	dout2_7	AT %QX1.6:	BOOL;
	su3_vent	AT %QX1.7:	BOOL;
	dout3_1	AT %QX2.0:	BOOL;

	lights_terminal1				AT %QB2:BYTE;

	spalnya_kontrazhur			AT %QX2.1:	BOOL; (*c*)
	spalnya_balkon				AT %QX2.2:	BOOL; (*c2*)
	dout3_4						AT %QX2.3:	BOOL;
	spalnya_kulbaba			AT %QX2.4:	BOOL;(*c3, c3a*)
	spalnya_kontrazhur_b		AT %QX2.5:	BOOL; (*c7*)
	spalnya_kontrazhur_l		AT %QX2.6:	BOOL; (*c4*)
	su3_stina					AT %QX2.7:	BOOL; (*c8*)
	(*dout4_1*)
	lights_terminal2				AT %QB3:BYTE;
	su3_pidsvitka 				AT %QX3.0:	BOOL;(*c10*)
	su3_bra						AT %QX3.1:	BOOL;(*c15*)
	su3_kontrazhur				AT %QX3.2:	BOOL;(*c9*)
	dytjacha					AT %QX3.3:	BOOL;(*c14*)
	su3_kontrazhur_k			AT %QX3.4:	BOOL; (*c11*)
	dytjacha_bra				AT %QX3.5:	BOOL; (*c15*)
	su3_lampa					AT %QX3.6:	BOOL; (*c12*)
	garderob					AT %QX3.7:	BOOL;
	(*dout5_1*)
	serverna					AT %QX4.0:	BOOL;
	bar							AT %QX4.1:	BOOL;(*c21*)
	korydor_skeli 				AT %QX4.2:	BOOL;(*c18*)
	choven						AT %QX4.3:	BOOL;(*c22*)
	korydor_svitlo				AT %QX4.4:	BOOL;(*c19*)
	fancoil_spalnya_low 			AT %QX4.5:	BOOL;
	korydor_lampa				AT %QX4.6:	BOOL;(*c20*)
	fancoil_spalnya_med			AT %QX4.7:	BOOL;
	(*dout6_1*)
	fancoil_spalnya_high			AT%QX5.0:BOOL;
	rozetky1					AT%QX5.1 :BOOL;
	fancoil_dytjacha_low			AT%QX5.2 :BOOL;
	rozetky2			 		AT%QX5.3 :BOOL;
	fancoil_dytjacha_med		AT%QX5.4:BOOL;
	rozetky3 					AT%QX5.5:BOOL;
	fancoil_dytjacha_high		AT%QX5.6:BOOL;
	rozetky4 					AT%QX5.7:BOOL;
	(*dout7_1*)
	rozetky5					AT%QX6.0:BOOL;
	tul_close 					AT%QX6.1 :BOOL;
	rozetky6	 				AT%QX6.2 :BOOL;
	tul_open	 				AT%QX6.3 :BOOL;
	shtory_close 				AT%QX6.4:BOOL;
	lift_down					AT%QX6.5:BOOL;
	shtory_open					AT%QX6.6:BOOL;
	lift_up	 					AT%QX6.7:BOOL;
(*dout8_1*)
	dytjacha_col 				AT%QX7.0:BOOL; (*тепла підлога*)
	serverna_col 				AT%QX7.1 :BOOL;
	freshbar_col 				AT%QX7.2 :BOOL;
	spalnya_col 					AT%QX7.3 :BOOL;
	korydor_col		 			AT%QX7.4:BOOL;
	su_col_pidloga 				AT%QX7.5:BOOL;
	su_col_stina					AT%QX7.6:BOOL;
	out88 AT%QX7.7:BOOL;
	out91 AT%QX8.0:BOOL;
	out92 AT%QX8.1 :BOOL;
	out93 AT%QX8.2 :BOOL;
	out94 AT%QX8.3 :BOOL;
	out95 AT%QX8.4:BOOL;
	out96 AT%QX8.5:BOOL;
	out97 AT%QX8.6:BOOL;
	out98 AT%QX8.7:BOOL;

	klapan_dytjacha		AT %QB10:	INT;
	klapan_spalnya		AT %QB12:	INT;
	KL4414_3_Out		AT %QB14:	INT;
	klapan_vitalnya		AT %QB16:	INT;
(*light sensors*)
	iLight_N			AT %IB28:INT;
	iLight_W			AT %IB30:INT;
	iLight_S			AT %IB32:INT;
	iLight_E			AT %IB34:INT;

	KL6301_IN_0 AT %IB4: ARRAY[1..24] OF BYTE;
	KL6301_OUT_0 AT %QB34: ARRAY[1..24] OF BYTE;

	iT_tambur	AT %IB36: INT;(*тепла підлога*)
	iT_su		AT %IB38: INT;(*тепла підлога*)
	iT_spalnya	AT %IB40: INT;(*тепла підлога*)
	iT_out			AT %IB42:INT; (*зовнішня температура*)

END_VAR

(* Data type *)
TYPE ROOM_HVAC :
STRUCT
	manual_mode:BOOL;
	heat_mode: USINT; (*1-cool, 2-heat, 3-fan*)
	heat_speed: USINT;

	cur_t:REAL;
	cur_t_ust,cur_t_ust_prev, t_ust_heat,	t_ust_cool:REAL;
	cooling_signal,heating_signal:BYTE;

	fancoil_speed:SINT;
	klapan:WORD;


	floor_heating:BOOL;
	floor_T	:REAL;
	floor_Sp	:REAL;

	zaslinka:BOOL;


END_STRUCT
END_TYPE

(* POU MAIN, ST *)
PROGRAM MAIN
VAR
	fbTimer: TON;
	fbRTC: RTC;
	i:INT;
	fbDarkTimeCorrection : TP;

	write1, write2, write4: BOOL;
	i2,j2,i1,j1, i4,j4: INT;
	repeat1, repeat2,repeat4:BOOL;


	init: BOOL;
	SpalnyaLiftToSafePos: BOOL;
	iSaidItsFuckingDARK	: BOOL;
END_VAR
IF init THEN
	SpalnyaLiftToSafePos:=TRUE;
	init:=FALSE;
END_IF

fbTimer(PT:=t#1s,IN:=NOT fbTimer.Q);

IF fbTimer.Q OR SYSTEMTASKINFOARR[1].firstCycle  THEN
	fbRTC;
END_IF

fbDarkTimeCorrection(IN:=iLight_N<1000 AND  iLight_W <1000 AND iLight_S <1000 AND iLight_E <1000, PT:=t#40m);
IF iLight_N<1000 AND  iLight_W <1000 AND iLight_S <1000 AND iLight_E <1000  AND NOT fbDarkTimeCorrection.q AND ( system_time.wHour>15 OR system_time.wHour<9)  THEN
	bDarkOutside:=TRUE OR iSaidItsFuckingDARK;
ELSE
	bDarkOutside:=FALSE OR iSaidItsFuckingDARK;
END_IF
(*EIB init*)
EIB;
(*Світло*)
Light;
Shtory;
(*климат*)
climate;
ADS_write;
ADS_Communication;

SpalnyaLiftToSafePos:=FALSE;
END_PROGRAM
ACTION ADS_write:
FOR i2:=0 TO (SIZEOF(data2floor))-1 DO
	IF data2floor[i2]<>data2floor_prev[i2]  THEN
		write2:=TRUE;
		EXIT;
	ELSE
		write2:=FALSE;
	END_IF
END_FOR


FOR i1:=0 TO (SIZEOF(data1floor))-1 DO
	IF data1floor[i1]<>data1floor_prev[i1]  THEN
		write1:=TRUE;
		EXIT;
	ELSE
		write1:=FALSE;
	END_IF
END_FOR


FOR i4:=0 TO (SIZEOF(data_derevo))-1 DO
	IF data_derevo[i4]<>data_derevo_prev[i4]  THEN
		write4:=TRUE;
		EXIT;
	ELSE
		write4:=FALSE;
	END_IF
END_FOR

FOR j1:=0 TO (SIZEOF(data1floor))-1 DO
	data1floor_prev[j1]:=data1floor[j1];
END_FOR

FOR j2:=0 TO (SIZEOF(data2floor))-1 DO
	data2floor_prev[j2]:=data2floor[j2];
END_FOR

FOR j4:=0 TO (SIZEOF(data_derevo))-1 DO
	data_derevo_prev[j4]:=data_derevo[j4];
END_FOR
END_ACTION

(* POU EIB, ST *)
PROGRAM EIB
VAR
	i:INT:=0;
	POWER: EIB_BIT_REC;
	fb_temp_read: EIB_2OCTET_FLOAT_REC;
	fb_read_heating_mode:EIB_BIT_REC;
	fb_req_heating_mode:EIB_READ_SEND;
	fb_setpoint_read:EIB_8BIT_UNSIGN_REC;
	setpoint_vitalnya_dpt4,	setpoint_kino_dpt4,	setpoint_studio_dpt4,	setpoint_kabinet_dpt4,	setpoint_dytjacha_dpt4,	setpoint_spalnya_dpt4:REAL;
	fanspeed_dpt4:REAL;



	fb_actual_setpoint_read:EIB_2OCTET_FLOAT_REC;
	fb_actual_setpoint_send:EIB_2OCTET_FLOAT_SEND;
	fb_out_temp_send:EIB_2OCTET_FLOAT_SEND;
	fb_setpoint_switch_send:EIB_BIT_SEND_EX;

	fb_start_delay:TP;

	fb_vitalnya_FCU_cooling_ctrl_sig_rec: EIB_8BIT_UNSIGN_REC;
	fb_kino_FCU_cooling_ctrl_sig_rec: EIB_8BIT_UNSIGN_REC;
	fb_kabinet_FCU_cooling_ctrl_sig_rec: EIB_8BIT_UNSIGN_REC;
	fb_dytjacha_FCU_cooling_ctrl_sig_rec: EIB_8BIT_UNSIGN_REC;
	fb_spalnya_FCU_cooling_ctrl_sig_rec: EIB_8BIT_UNSIGN_REC;

	fb_vitalnya_FCU_heating_ctrl_sig_rec: EIB_8BIT_UNSIGN_REC;
	fb_kino_FCU_heating_ctrl_sig_rec: EIB_8BIT_UNSIGN_REC;
	fb_kabinet_FCU_heating_ctrl_sig_rec: EIB_8BIT_UNSIGN_REC;
	fb_dytjacha_FCU_heating_ctrl_sig_rec: EIB_8BIT_UNSIGN_REC;
	fb_spalnya_FCU_heating_ctrl_sig_rec: EIB_8BIT_UNSIGN_REC;

	fb_vitalnya_FCU_fan_speed_send: EIB_8BIT_UNSIGN_SEND;
	fb_kino_FCU_fan_speed_send: EIB_8BIT_UNSIGN_SEND;
	fb_dytjacha_FCU_fan_speed_send: EIB_8BIT_UNSIGN_SEND;
	fb_spalnya_FCU_fan_speed_send: EIB_8BIT_UNSIGN_SEND;
	fb_kabinet_FCU_fan_speed_send: EIB_8BIT_UNSIGN_SEND;

	fb_vitalnya_damper_ctrl_rec: EIB_BIT_REC;
	fb_kino_damper_ctrl_rec: EIB_BIT_REC;
	fb_kabinet_damper_ctrl_rec: EIB_BIT_REC;
	fb_dytjacha_damper_ctrl_rec: EIB_BIT_REC;
	fb_spalnya_damper_ctrl_rec: EIB_BIT_REC;



	fb_eib_time_rec: EIB_TIME_REC;
	fb_eib_date_rec: EIB_DATE_REC;
	fb_eib_dark_outside_rec: EIB_BIT_REC;
	fb_beckhoff_twillight_send: EIB_BIT_SEND;

	(*eib_twillight_eib_addr: EIB_GROUP_ADDR := (MAIN:=1,SUB_MAIN:=3,NUMBER:=14);*)
	b_eib_twillight: BOOL;
	fb_eib_twillight_send: EIB_BIT_SEND;
	fb_eib_twillight_rec: EIB_BIT_REC;
	beckhoff_twillight_eib_addr: EIB_GROUP_ADDR := (MAIN:=1,SUB_MAIN:=3,NUMBER:=13);

	eib_send_mode_floor1: INT;
	eib_send_cyclical_start_floor1: BOOL := TRUE;
	eib_send_mode_floor2: INT;
	eib_send_cyclical_start_floor2: BOOL := TRUE;
	eib_send_mode_floor3: INT;
	eib_send_cyclical_start_floor3: BOOL := TRUE;
	eib_send_mode_floor4: INT;
	eib_send_cyclical_start_floor4: BOOL := TRUE;

	floors:INT;
	fb_sending_floor_order:CTU;
	fb_heartbeat_timer:TON;
	fb_sending_time_frame:TOF;

	fbNightLightTimer:		TP;



END_VAR
fb_start_delay(IN:=  SYSTEMTASKINFOARR[1].firstCycle, PT:=t#60s);
fb_req_heating_mode.bRead:=FALSE;
IF  fb_start_delay.Q THEN
	fb_req_heating_mode(group_address:=heating_mode_addr, str_Rec:=fb_kl6301_0.str_Data_Rec, bread:=fb_start_delay.Q);
END_IF;
fb_read_heating_mode(strData_Rec:=fb_KL6301_0.str_Data_Rec, Group_Address:=heating_mode_addr, bdata=>heating_mode);
(*EIB*)
fb_heartbeat_timer(in:=NOT  fb_heartbeat_timer.Q, pt:=t#30m);
fb_sending_time_frame(in:=fb_heartbeat_timer.Q, pt:=t#50ms);
fb_sending_floor_order(cu:=fb_heartbeat_timer.Q, pv:=4,reset:=fb_sending_floor_order.CV >4, CV=>floors);

eib_send_mode_floor1:=2;
eib_send_mode_floor2:=2;
eib_send_mode_floor3:=2;
eib_send_mode_floor4:=2;

CASE floors OF
1:
	eib_send_mode_floor1:=2*BOOL_TO_INT(NOT (fb_sending_time_frame.Q)); (*0-manual*)
	IF fb_heartbeat_timer.Q THEN
		eib_send_cyclical_start_floor1:=FALSE;
	ELSE
		eib_send_cyclical_start_floor1:=TRUE;
	END_IF
2:
	eib_send_mode_floor2:=2*BOOL_TO_INT(NOT (fb_sending_time_frame.Q)); (*0-manual*)
	IF fb_heartbeat_timer.Q THEN
		eib_send_cyclical_start_floor2:=FALSE;
	ELSE
		eib_send_cyclical_start_floor2:=TRUE;
	END_IF
3:
	eib_send_mode_floor3:=2*BOOL_TO_INT(NOT (fb_sending_time_frame.Q)); (*0-manual*)
	IF fb_heartbeat_timer.Q THEN
		eib_send_cyclical_start_floor3:=FALSE;
	ELSE
		eib_send_cyclical_start_floor3:=TRUE;
	END_IF
4:
	eib_send_mode_floor4:=2*BOOL_TO_INT(NOT (fb_sending_time_frame.Q)); (*0-manual*)
	IF fb_heartbeat_timer.Q THEN
		eib_send_cyclical_start_floor4:=FALSE;
	ELSE
		eib_send_cyclical_start_floor4:=TRUE;
	END_IF
END_CASE


fb_KL6301_0.iMode:=1;
CASE i OF
0:	(* EIB Address 2.3.4 *)
	fb_KL6301_0.EIB_PHYS_ADDR.Area:=1;
	fb_KL6301_0.EIB_PHYS_ADDR.Line:=1;
	fb_KL6301_0.EIB_PHYS_ADDR.Device:=1;
	(* Filter 1 *)
	fb_KL6301_0.EIB_GROUP_FILTER[1].GROUP_ADDR.MAIN:=1;
	fb_KL6301_0.EIB_GROUP_FILTER[1].GROUP_ADDR.SUB_MAIN:=1;
	fb_KL6301_0.EIB_GROUP_FILTER[1].GROUP_ADDR.NUMBER:=0;
	fb_KL6301_0.EIB_GROUP_FILTER[1].GROUP_LEN:=31;
	(* Filter 2*)
	fb_KL6301_0.EIB_GROUP_FILTER[2].GROUP_ADDR.MAIN:=1;
	fb_KL6301_0.EIB_GROUP_FILTER[2].GROUP_ADDR.SUB_MAIN:=2;
	fb_KL6301_0.EIB_GROUP_FILTER[2].GROUP_ADDR.NUMBER:=0;
	fb_KL6301_0.EIB_GROUP_FILTER[2].GROUP_LEN:=31;
	(* Filter 3*)
	fb_KL6301_0.EIB_GROUP_FILTER[3].GROUP_ADDR.MAIN:=1;
	fb_KL6301_0.EIB_GROUP_FILTER[3].GROUP_ADDR.SUB_MAIN:=3;
	fb_KL6301_0.EIB_GROUP_FILTER[3].GROUP_ADDR.NUMBER:=0;
	fb_KL6301_0.EIB_GROUP_FILTER[3].GROUP_LEN:=31;
	(* Filter 4 *)
	fb_KL6301_0.EIB_GROUP_FILTER[4].GROUP_ADDR.MAIN:=1;
	fb_KL6301_0.EIB_GROUP_FILTER[4].GROUP_ADDR.SUB_MAIN:=4;
	fb_KL6301_0.EIB_GROUP_FILTER[4].GROUP_ADDR.NUMBER:=0;
	fb_KL6301_0.EIB_GROUP_FILTER[4].GROUP_LEN:=31;
	(* Filter 5*)
	fb_KL6301_0.EIB_GROUP_FILTER[5].GROUP_ADDR.MAIN:=1;
	fb_KL6301_0.EIB_GROUP_FILTER[5].GROUP_ADDR.SUB_MAIN:=5;
	fb_KL6301_0.EIB_GROUP_FILTER[5].GROUP_ADDR.NUMBER:=0;
	fb_KL6301_0.EIB_GROUP_FILTER[5].GROUP_LEN:=31;
	(* Filter 6*)
	fb_KL6301_0.EIB_GROUP_FILTER[6].GROUP_ADDR.MAIN:=1;
	fb_KL6301_0.EIB_GROUP_FILTER[6].GROUP_ADDR.SUB_MAIN:=6;
	fb_KL6301_0.EIB_GROUP_FILTER[6].GROUP_ADDR.NUMBER:=0;
	fb_KL6301_0.EIB_GROUP_FILTER[6].GROUP_LEN:=31;
	(* Filter 7*)
	fb_KL6301_0.EIB_GROUP_FILTER[7].GROUP_ADDR.MAIN:=1;
	fb_KL6301_0.EIB_GROUP_FILTER[7].GROUP_ADDR.SUB_MAIN:=7;
	fb_KL6301_0.EIB_GROUP_FILTER[7].GROUP_ADDR.NUMBER:=0;
	fb_KL6301_0.EIB_GROUP_FILTER[7].GROUP_LEN:=31;
(*	(* Filter 8*)
	fb_KL6301_0.EIB_GROUP_FILTER[8].GROUP_ADDR.MAIN:=1;
	fb_KL6301_0.EIB_GROUP_FILTER[8].GROUP_ADDR.SUB_MAIN:=8;
	fb_KL6301_0.EIB_GROUP_FILTER[8].GROUP_ADDR.NUMBER:=0;
	fb_KL6301_0.EIB_GROUP_FILTER[8].GROUP_LEN:=31;*)

	fb_KL6301_0.bActivate :=TRUE; 	(*Start EIB Functionblock*)
	IF fb_KL6301_0.bReady THEN	(*Wait until the fb is ready *)
		IF NOT fb_KL6301_0.bError THEN
			i:=1;  (* EIB functionblock is now ready to send and receive *)
		ELSE
			i:=100; (* EIB ERROR*)
		END_IF
	END_IF
1:	;
100:	;(*ERROR EIB*)
END_CASE

fb_KL6301_0(
	idx:=1,								(* for every KL6301 an other idx number
										Example KL6301 terminal 1 - idx=1 , KL6301 termnal 2 -idx=3,... max. 64 *)
	KL6301_IN:=KL6301_IN_0,				(* Terminal variable - address IN *)
	KL6301_OUT:=KL6301_OUT_0 );			(* Terminal variable - address OUT *)



eibPort_climate;
floor1;
floor2;
floor3;
derevo;
central_lights;
timers;
END_PROGRAM
ACTION central_lights:
(*fb_floor1_lights_read(strData_Rec:=fb_KL6301_0.str_Data_Rec, Group_Address:=lights_out_floor1_eib_addr );
IF NOT  fb_floor1_lights_read.bDataReceive AND NOT fb_floor1_lights_read.bData THEN
	floor1_lights:= FALSE;
ELSE*)

	IF data1floor[100] > 0 OR data1floor[101] > 0  THEN
		floor1_lights :=TRUE;
	ELSE
		floor1_lights:=FALSE;
	END_IF
(*END_IF*)
(*
fb_floor2_lights_read(strData_Rec:=fb_KL6301_0.str_Data_Rec, Group_Address:=lights_out_floor2_eib_addr );
IF NOT  fb_floor2_lights_read.bDataReceive AND NOT fb_floor2_lights_read.bData THEN
	floor2_lights:= FALSE;
ELSE*)

	IF data2floor[100] > 0 OR data2floor[101] > 0  OR data2floor[102] > 0 THEN
		floor2_lights :=TRUE;
	ELSE
		floor2_lights:=FALSE;
	END_IF
(*END_IF*)
(*
fb_floor3_lights_read(strData_Rec:=fb_KL6301_0.str_Data_Rec, Group_Address:=lights_out_floor3_eib_addr );
IF NOT  fb_floor3_lights_read.bDataReceive AND NOT fb_floor3_lights_read.bData THEN
	floor3_lights:= FALSE;
ELSE*)

	IF lights_terminal1 > 0 OR lights_terminal2 >0 OR bar OR korydor_skeli OR korydor_svitlo OR choven OR serverna THEN
		floor3_lights := TRUE;
	ELSE
		floor3_lights:=FALSE;
	END_IF
(*END_IF*)

(*fb_derevo_lights_read(strData_Rec:=fb_KL6301_0.str_Data_Rec, Group_Address:=lights_out_derevo_eib_addr );
IF (NOT  fb_derevo_lights_read.bDataReceive) AND (NOT fb_derevo_lights_read.bData) THEN
	derevo_lights:= FALSE;
ELSE*)

	IF data_derevo[100] > 0 OR data_derevo[101] > 0 OR data_derevo[102] > 0 THEN
		derevo_lights :=TRUE;
	ELSE
		derevo_lights:=FALSE;
	END_IF
(*END_IF*)

(*fb_main_house_lights_read(strData_Rec:=fb_KL6301_0.str_Data_Rec, Group_Address:=lights_out_main_house_eib_addr );
IF NOT  fb_main_house_lights_read.bDataReceive AND NOT fb_main_house_lights_read.bData THEN
	main_house_lights:= FALSE;
ELSE*)

	IF floor1_lights OR floor2_lights OR floor3_lights THEN
		main_house_lights:=TRUE;
	ELSE
		main_house_lights:=FALSE;
	END_IF
(*END_IF*)

(*fb_all_lights_read(strData_Rec:=fb_KL6301_0.str_Data_Rec, Group_Address:=lights_out_all_eib_addr );
IF NOT  fb_all_lights_read.bDataReceive AND NOT fb_all_lights_read.bData THEN
	main_house_lights:= FALSE;
ELSE*)
	IF main_house_lights OR derevo_lights THEN
		all_lights:=TRUE;
	ELSE
		all_lights:=FALSE;
	END_IF
(*END_IF*)


fb_floor1_lights_send_status_ex(imode:=2, bStart:=TRUE, str_Rec:=fb_KL6301_0.str_Data_Rec, bData:=floor1_lights,  Group_Address:=lights_out_floor1_eib_addr);
fb_floor2_lights_send_status_ex(imode:=2, bStart:=TRUE, str_Rec:=fb_KL6301_0.str_Data_Rec, bData:=floor2_lights,  Group_Address:=lights_out_floor2_eib_addr);
fb_floor3_lights_send_status_ex(imode:=2, bStart:=TRUE, str_Rec:=fb_KL6301_0.str_Data_Rec, bData:=floor3_lights,  Group_Address:=lights_out_floor3_eib_addr);
fb_derevo_lights_send_status_ex(imode:=2, bStart:=TRUE, str_Rec:=fb_KL6301_0.str_Data_Rec, bData:=derevo_lights,  Group_Address:=lights_out_derevo_eib_addr);
fb_main_house_lights_send_status_ex(imode:=2, bStart:=TRUE, str_Rec:=fb_KL6301_0.str_Data_Rec, bData:=main_house_lights,  Group_Address:=lights_out_main_house_eib_addr);
fb_all_lights_send_status_ex(imode:=2, bStart:=TRUE, str_Rec:=fb_KL6301_0.str_Data_Rec, bData:=all_lights,  Group_Address:=lights_out_all_eib_addr);
END_ACTION
ACTION derevo:
data_derevo[0].0:=bDarkOutside;

data_derevo[4]:=WORD_TO_BYTE(system_time.wHour);
data_derevo[5]:=WORD_TO_BYTE(system_time.wMinute);

MEMCPY(ADR(data_derevo[10] ), ADR(OAT), SIZEOF(OAT));


fb_derevo_vidpochynok1_read(strData_Rec:=fb_KL6301_0.str_Data_Rec, Group_Address:=derevo_vidpochynok1_adr);
IF NOT  fb_derevo_vidpochynok1_read.bDataReceive THEN
	data_derevo[100].0:= fb_derevo_vidpochynok1_read.bdata;
END_IF

fb_derevo_vidpochynok2_read(strData_Rec:=fb_KL6301_0.str_Data_Rec, Group_Address:=derevo_vidpochynok2_adr);
IF NOT  fb_derevo_vidpochynok2_read.bDataReceive THEN
	data_derevo[100].1:= fb_derevo_vidpochynok2_read.bdata;
END_IF

fb_derevo_veranda_read(strData_Rec:=fb_KL6301_0.str_Data_Rec, Group_Address:=derevo_veranda_adr);
IF NOT  fb_derevo_veranda_read.bDataReceive THEN
	data_derevo[100].2:= fb_derevo_veranda_read.bdata;
END_IF

fb_derevo_veranda_zovn_read(strData_Rec:=fb_KL6301_0.str_Data_Rec, Group_Address:=derevo_veranda_zovn_adr);
IF NOT  fb_derevo_veranda_zovn_read.bDataReceive THEN
	data_derevo[100].3:=fb_derevo_veranda_zovn_read.bdata;
END_IF

fb_derevo_vhid_zovn_read(strData_Rec:=fb_KL6301_0.str_Data_Rec, Group_Address:=derevo_vhid_zovn_adr);
IF NOT  fb_derevo_vhid_zovn_read.bDataReceive THEN
	data_derevo[100].4:= fb_derevo_vhid_zovn_read.bdata;
END_IF

fb_derevo_sauna_read(strData_Rec:=fb_KL6301_0.str_Data_Rec, Group_Address:=derevo_sauna_adr);
IF NOT  fb_derevo_sauna_read.bDataReceive THEN
	data_derevo[100].5:= fb_derevo_sauna_read.bdata;
END_IF

fb_derevo_vhid_read(strData_Rec:=fb_KL6301_0.str_Data_Rec, Group_Address:=derevo_vhid_adr);
IF NOT  fb_derevo_vhid_read.bDataReceive THEN
	data_derevo[100].6:= fb_derevo_vhid_read.bdata;
END_IF

fb_derevo_kotel_read(strData_Rec:=fb_KL6301_0.str_Data_Rec, Group_Address:=derevo_kotel_adr);
IF NOT  fb_derevo_kotel_read.bDataReceive THEN
	data_derevo[100].7:= fb_derevo_kotel_read.bdata;
END_IF

fb_derevo_korydor_read(strData_Rec:=fb_KL6301_0.str_Data_Rec, Group_Address:=derevo_korydor_adr );
IF NOT  fb_derevo_korydor_read.bDataReceive THEN
	data_derevo[101].0:= fb_derevo_korydor_read.bdata;
END_IF
fb_derevo_sinna_read(strData_Rec:=fb_KL6301_0.str_Data_Rec, Group_Address:=derevo_sinna_adr );
IF NOT  fb_derevo_sinna_read.bDataReceive THEN
	data_derevo[101].1:= fb_derevo_sinna_read.bdata;
END_IF
fb_derevo_hamam_read(strData_Rec:=fb_KL6301_0.str_Data_Rec, Group_Address:=derevo_hamam_adr );
IF NOT  fb_derevo_hamam_read.bDataReceive THEN
	data_derevo[101].2:= fb_derevo_hamam_read.bdata;
END_IF
fb_derevo_kuhnya_read(strData_Rec:=fb_KL6301_0.str_Data_Rec, Group_Address:=derevo_kuhnya_adr );
IF NOT  fb_derevo_kuhnya_read.bDataReceive THEN
	data_derevo[101].3:= fb_derevo_kuhnya_read.bdata;
END_IF
fb_derevo_bassein1_read(strData_Rec:=fb_KL6301_0.str_Data_Rec, Group_Address:=derevo_bassein1_adr );
IF NOT  fb_derevo_bassein1_read.bDataReceive THEN
	data_derevo[101].4:= fb_derevo_bassein1_read.bdata;
END_IF
fb_derevo_bassein_lampa_read(strData_Rec:=fb_KL6301_0.str_Data_Rec, Group_Address:=derevo_bassein_lampa_adr );
IF NOT  fb_derevo_bassein_lampa_read.bDataReceive THEN
	data_derevo[101].5:= fb_derevo_bassein_lampa_read.bdata;
END_IF
fb_derevo_spalnya2_read(strData_Rec:=fb_KL6301_0.str_Data_Rec, Group_Address:=derevo_spalnya2_adr);
IF NOT  fb_derevo_spalnya2_read.bDataReceive THEN
	data_derevo[101].6:= fb_derevo_spalnya2_read.bdata;
END_IF
fb_derevo_terassa_read(strData_Rec:=fb_KL6301_0.str_Data_Rec, Group_Address:=derevo_terassa_adr);
IF NOT  fb_derevo_terassa_read.bDataReceive THEN
	data_derevo[101].7:= fb_derevo_terassa_read.bdata;
END_IF
fb_derevo_dush_read(strData_Rec:=fb_KL6301_0.str_Data_Rec, Group_Address:=derevo_dush_adr );
IF NOT  fb_derevo_dush_read.bDataReceive THEN
	data_derevo[102].0:= fb_derevo_dush_read.bdata;
END_IF
fb_derevo_wc_read(strData_Rec:=fb_KL6301_0.str_Data_Rec, Group_Address:=derevo_wc_adr );
IF NOT  fb_derevo_wc_read.bDataReceive THEN
	data_derevo[102].1:= fb_derevo_wc_read.bdata;
END_IF
fb_derevo_spalnya_verh_read(strData_Rec:=fb_KL6301_0.str_Data_Rec, Group_Address:=derevo_spalnya_verh_adr );
IF NOT  fb_derevo_spalnya_verh_read.bDataReceive THEN
	data_derevo[102].2:= fb_derevo_spalnya_verh_read.bdata;
END_IF
fb_derevo_spalnya1_read(strData_Rec:=fb_KL6301_0.str_Data_Rec, Group_Address:=derevo_spalnya1_adr );
IF NOT  fb_derevo_spalnya1_read.bDataReceive THEN
	data_derevo[102].3:= fb_derevo_spalnya1_read.bdata;
END_IF
fb_derevo_spalnya_su_read(strData_Rec:=fb_KL6301_0.str_Data_Rec, Group_Address:=derevo_spalnya_su_adr );
IF NOT  fb_derevo_spalnya_su_read.bDataReceive THEN
	data_derevo[102].4:= fb_derevo_spalnya_su_read.bdata;
END_IF
fb_derevo_garderob_read(strData_Rec:=fb_KL6301_0.str_Data_Rec, Group_Address:=derevo_garderob_adr );
IF NOT  fb_derevo_garderob_read.bDataReceive THEN
	data_derevo[102].5:= fb_derevo_garderob_read.bdata;
END_IF

fb_derevo_dush2_read(strData_Rec:=fb_KL6301_0.str_Data_Rec, Group_Address:=derevo_dush2_adr );
IF NOT  fb_derevo_dush2_read.bDataReceive THEN
	data_derevo[102].6:= fb_derevo_dush2_read.bdata;
END_IF

fb_derevo_okno_basseina_read(strData_Rec:=fb_KL6301_0.str_Data_Rec, Group_Address:=derevo_okno_basseina_adr );
IF NOT  fb_derevo_okno_basseina_read.bDataReceive THEN
	data_derevo[103].0:= fb_derevo_okno_basseina_read.bdata;
END_IF
(*sending*)

fb_derevo_vidpochynok1_send_status_ex(imode:=eib_send_mode_floor4, bStart:=eib_send_cyclical_start_floor4, str_Rec:=fb_KL6301_0.str_Data_Rec, bData:=derevo_vidpochynok1,  Group_Address:=derevo_vidpochynok1_status_adr);
fb_derevo_vidpochynok2_send_status_ex(imode:=eib_send_mode_floor4, bStart:=eib_send_cyclical_start_floor4, str_Rec:=fb_KL6301_0.str_Data_Rec, bData:=derevo_vidpochynok2,  Group_Address:=derevo_vidpochynok2_status_adr);
fb_derevo_veranda_send_status_ex(imode:=eib_send_mode_floor4, bStart:=eib_send_cyclical_start_floor4, str_Rec:=fb_KL6301_0.str_Data_Rec, bData:=derevo_veranda,  Group_Address:=derevo_veranda_status_adr);
fb_derevo_veranda_zovn_send_status_ex(imode:=eib_send_mode_floor4, bStart:=eib_send_cyclical_start_floor4, str_Rec:=fb_KL6301_0.str_Data_Rec, bData:=derevo_veranda_zovn,  Group_Address:=derevo_veranda_zovn_status_adr);
fb_derevo_sauna_send_status_ex(imode:=eib_send_mode_floor4, bStart:=eib_send_cyclical_start_floor4, str_Rec:=fb_KL6301_0.str_Data_Rec, bData:=derevo_sauna,  Group_Address:=derevo_sauna_status_adr);
fb_derevo_vhid_zovn_send_status_ex(imode:=eib_send_mode_floor4, bStart:=eib_send_cyclical_start_floor4, str_Rec:=fb_KL6301_0.str_Data_Rec, bData:=derevo_vhid_zovn,  Group_Address:=derevo_vhid_zovn_status_adr);
fb_derevo_vhid_send_status_ex(imode:=eib_send_mode_floor4, bStart:=eib_send_cyclical_start_floor4, str_Rec:=fb_KL6301_0.str_Data_Rec, bData:=derevo_vhid,  Group_Address:=derevo_vhid_status_adr);
fb_derevo_kotel_send_status_ex(imode:=eib_send_mode_floor4, bStart:=eib_send_cyclical_start_floor4, str_Rec:=fb_KL6301_0.str_Data_Rec, bData:=derevo_kotel,  Group_Address:=derevo_kotel_status_adr);
fb_derevo_korydor_send_status_ex(imode:=eib_send_mode_floor4, bStart:=eib_send_cyclical_start_floor4, str_Rec:=fb_KL6301_0.str_Data_Rec, bData:=derevo_korydor,  Group_Address:=derevo_korydor_status_adr);
fb_derevo_sinna_send_status_ex(imode:=eib_send_mode_floor4, bStart:=eib_send_cyclical_start_floor4, str_Rec:=fb_KL6301_0.str_Data_Rec, bData:=derevo_sinna,  Group_Address:=derevo_sinna_status_adr);
fb_derevo_hamam_send_status_ex(imode:=eib_send_mode_floor4, bStart:=eib_send_cyclical_start_floor4, str_Rec:=fb_KL6301_0.str_Data_Rec, bData:=derevo_hamam,  Group_Address:=derevo_hamam_status_adr);
fb_derevo_kuhnya_send_status_ex(imode:=eib_send_mode_floor4, bStart:=eib_send_cyclical_start_floor4, str_Rec:=fb_KL6301_0.str_Data_Rec, bData:=derevo_kuhnya,  Group_Address:=derevo_kuhnya_status_adr);
fb_derevo_bassein1_send_status_ex(imode:=eib_send_mode_floor4, bStart:=eib_send_cyclical_start_floor4, str_Rec:=fb_KL6301_0.str_Data_Rec, bData:=derevo_bassein1,  Group_Address:=derevo_bassein1_status_adr);
fb_derevo_bassein_lampa_send_status_ex(imode:=eib_send_mode_floor4, bStart:=eib_send_cyclical_start_floor4, str_Rec:=fb_KL6301_0.str_Data_Rec, bData:=derevo_bassein_lampa,  Group_Address:=derevo_bassein_lampa_status_adr);
fb_derevo_spalnya2_send_status_ex(imode:=eib_send_mode_floor4, bStart:=eib_send_cyclical_start_floor4, str_Rec:=fb_KL6301_0.str_Data_Rec, bData:=derevo_spalnya2,  Group_Address:=derevo_spalnya2_status_adr);
fb_derevo_terassa_send_status_ex(imode:=eib_send_mode_floor4, bStart:=eib_send_cyclical_start_floor4, str_Rec:=fb_KL6301_0.str_Data_Rec, bData:=derevo_terassa,  Group_Address:=derevo_terassa_status_adr);
fb_derevo_dush_send_status_ex(imode:=eib_send_mode_floor4, bStart:=eib_send_cyclical_start_floor4, str_Rec:=fb_KL6301_0.str_Data_Rec, bData:=derevo_dush,  Group_Address:=derevo_dush_status_adr);
fb_derevo_wc_send_status_ex(imode:=eib_send_mode_floor4, bStart:=eib_send_cyclical_start_floor4, str_Rec:=fb_KL6301_0.str_Data_Rec, bData:=derevo_wc,  Group_Address:=derevo_wc_status_adr);
fb_derevo_spalnya_verh_send_status_ex(imode:=eib_send_mode_floor4, bStart:=eib_send_cyclical_start_floor4, str_Rec:=fb_KL6301_0.str_Data_Rec, bData:=derevo_spalnya_verh,  Group_Address:=derevo_spalnya_verh_status_adr);
fb_derevo_spalnya1_send_status_ex(imode:=eib_send_mode_floor4, bStart:=eib_send_cyclical_start_floor4, str_Rec:=fb_KL6301_0.str_Data_Rec, bData:=derevo_spalnya1,  Group_Address:=derevo_spalnya1_status_adr);
fb_derevo_spalnya_su_send_status_ex(imode:=eib_send_mode_floor4, bStart:=eib_send_cyclical_start_floor4, str_Rec:=fb_KL6301_0.str_Data_Rec, bData:=derevo_spalnya_su,  Group_Address:=derevo_spalnya_su_status_adr);
fb_derevo_garderob_send_status_ex(imode:=eib_send_mode_floor4, bStart:=eib_send_cyclical_start_floor4, str_Rec:=fb_KL6301_0.str_Data_Rec, bData:=derevo_garderob,  Group_Address:=derevo_garderob_status_adr);
fb_derevo_dush2_send_status_ex(imode:=eib_send_mode_floor4, bStart:=eib_send_cyclical_start_floor4, str_Rec:=fb_KL6301_0.str_Data_Rec, bData:=derevo_dush2,  Group_Address:=derevo_dush2_status_adr);
fb_derevo_okno_basseina_send_status_ex(imode:=eib_send_mode_floor4, bStart:=eib_send_cyclical_start_floor4, str_Rec:=fb_KL6301_0.str_Data_Rec, bData:=derevo_okno_basseina,  Group_Address:=derevo_okno_basseina_status_adr);

IF fb_derevo_vidpochynok1_send_status_ex.bBusy OR fb_heartbeat_timer.Q   THEN
	data_derevo[100].0:=derevo_vidpochynok1;
END_IF

IF fb_derevo_vidpochynok2_send_status_ex.bBusy OR fb_heartbeat_timer.Q  THEN
	data_derevo[100].1:=derevo_vidpochynok2;
END_IF

IF fb_derevo_veranda_send_status_ex.bBusy OR fb_heartbeat_timer.Q  THEN
	data_derevo[100].2:=derevo_veranda;
END_IF

IF fb_derevo_veranda_zovn_send_status_ex.bBusy OR fb_heartbeat_timer.Q    THEN
	data_derevo[100].3:=derevo_veranda_zovn;
END_IF

IF fb_derevo_vhid_zovn_send_status_ex.bBusy OR fb_heartbeat_timer.Q  THEN
	data_derevo[100].4:=derevo_vhid_zovn;
END_IF

IF fb_derevo_sauna_send_status_ex.bBusy OR fb_heartbeat_timer.Q  THEN
	data_derevo[100].5:=derevo_sauna;
END_IF

IF fb_derevo_vhid_send_status_ex.bBusy OR fb_heartbeat_timer.Q  THEN
	data_derevo[100].6:=derevo_vhid;
END_IF

IF fb_derevo_kotel_send_status_ex.bBusy OR fb_heartbeat_timer.Q  THEN
	data_derevo[100].7:=derevo_kotel;
END_IF

IF fb_derevo_korydor_send_status_ex.bBusy OR fb_heartbeat_timer.Q  THEN
	data_derevo[101].0:=derevo_korydor;
END_IF

IF fb_derevo_sinna_send_status_ex.bBusy OR fb_heartbeat_timer.Q  THEN
	data_derevo[101].1:=derevo_sinna;
END_IF

IF fb_derevo_hamam_send_status_ex.bBusy OR fb_heartbeat_timer.Q  THEN
	data_derevo[101].2:=derevo_hamam;
END_IF

IF fb_derevo_kuhnya_send_status_ex.bBusy OR fb_heartbeat_timer.Q  THEN
	data_derevo[101].3:=derevo_kuhnya;
END_IF

IF fb_derevo_bassein1_send_status_ex.bBusy OR fb_heartbeat_timer.Q  THEN
	data_derevo[101].4:=derevo_bassein1;
END_IF

IF fb_derevo_bassein_lampa_send_status_ex.bBusy OR fb_heartbeat_timer.Q  THEN
	data_derevo[101].5:=derevo_bassein_lampa;
END_IF

IF fb_derevo_spalnya2_send_status_ex.bBusy OR fb_heartbeat_timer.Q  THEN
	data_derevo[101].6:=derevo_spalnya2;
END_IF

IF fb_derevo_terassa_send_status_ex.bBusy OR fb_heartbeat_timer.Q  THEN
	data_derevo[101].7:=derevo_terassa;
END_IF

IF fb_derevo_dush_send_status_ex.bBusy OR fb_heartbeat_timer.Q  THEN
	data_derevo[102].0:=derevo_dush;
END_IF

IF fb_derevo_wc_send_status_ex.bBusy OR fb_heartbeat_timer.Q  THEN
	data_derevo[102].1:=derevo_wc;
END_IF

IF fb_derevo_spalnya_verh_send_status_ex.bBusy OR fb_heartbeat_timer.Q  THEN
	data_derevo[102].2:=derevo_spalnya_verh;
END_IF

IF fb_derevo_spalnya1_send_status_ex.bBusy OR fb_heartbeat_timer.Q  THEN
	data_derevo[102].3:=derevo_spalnya1;
END_IF

IF fb_derevo_spalnya_su_send_status_ex.bBusy OR fb_heartbeat_timer.Q  THEN
	data_derevo[102].4:=derevo_spalnya_su;
END_IF

IF fb_derevo_garderob_send_status_ex.bBusy OR fb_heartbeat_timer.Q  THEN
	data_derevo[102].5:=derevo_garderob;
END_IF

IF fb_derevo_dush2_send_status_ex.bBusy OR fb_heartbeat_timer.Q  THEN
	data_derevo[102].6:=derevo_dush2;
END_IF

IF fb_derevo_okno_basseina_send_status_ex.bBusy OR fb_heartbeat_timer.Q  THEN
	data_derevo[103].0:=derevo_okno_basseina;
END_IF
END_ACTION
ACTION eibPort_climate:
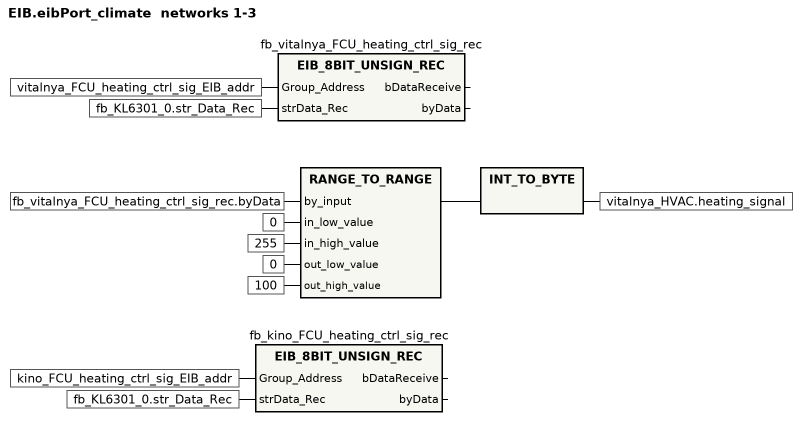
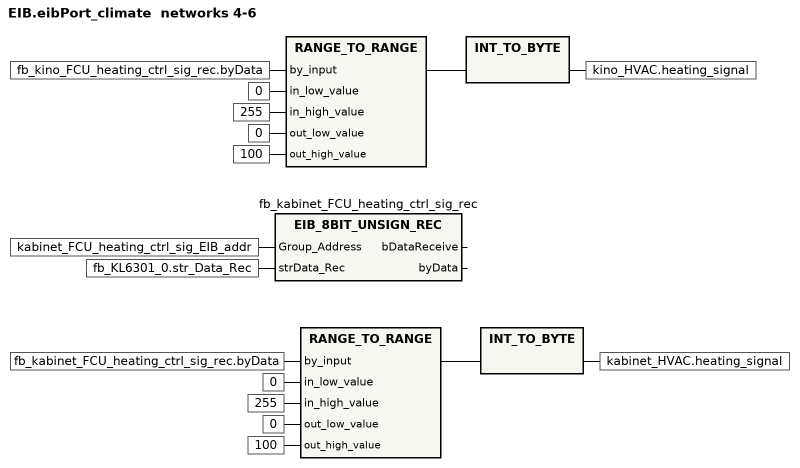
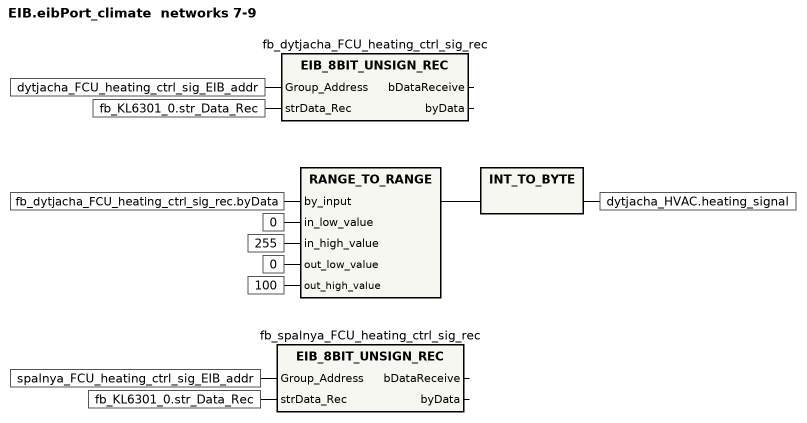
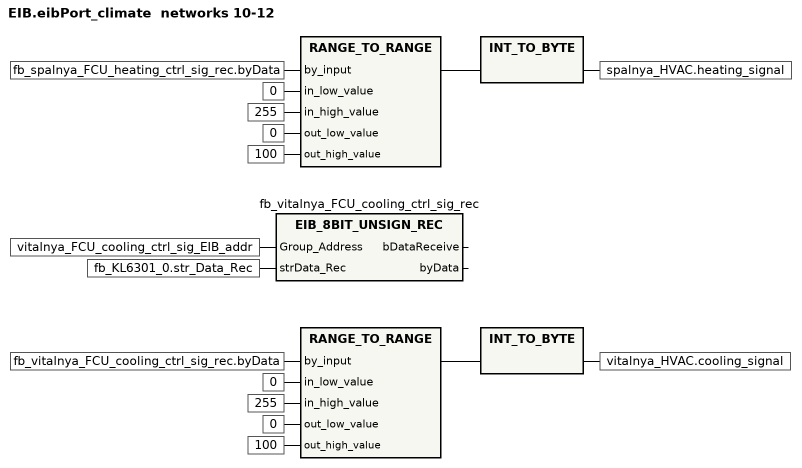
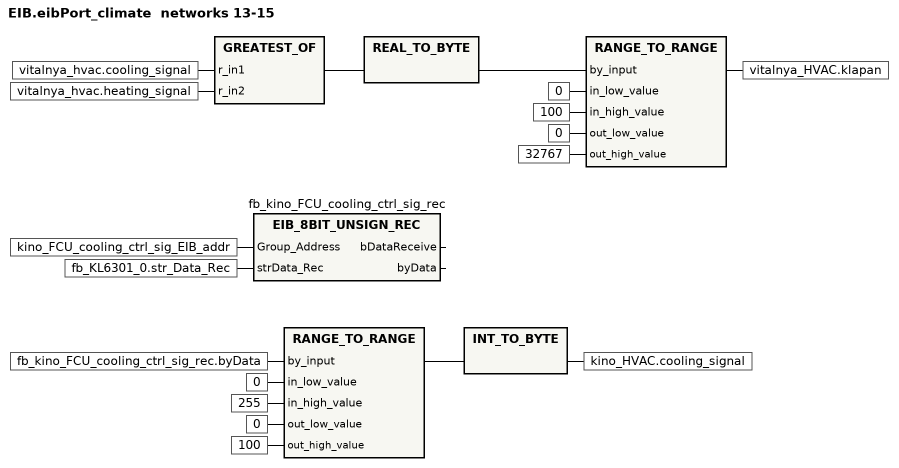
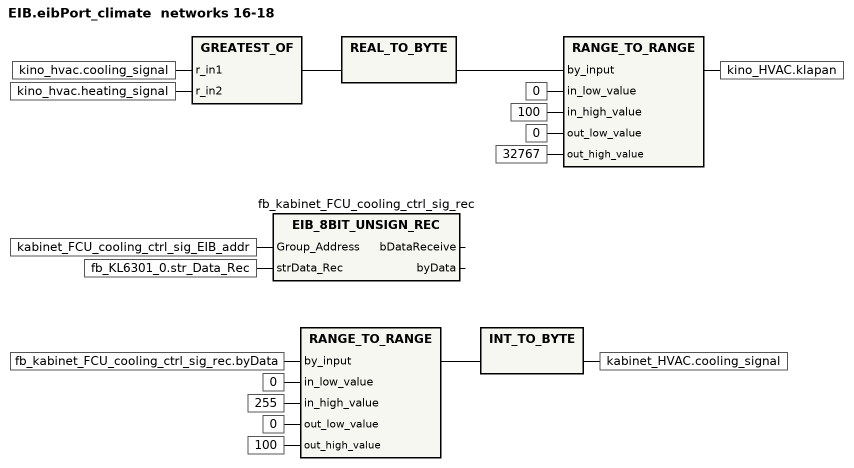
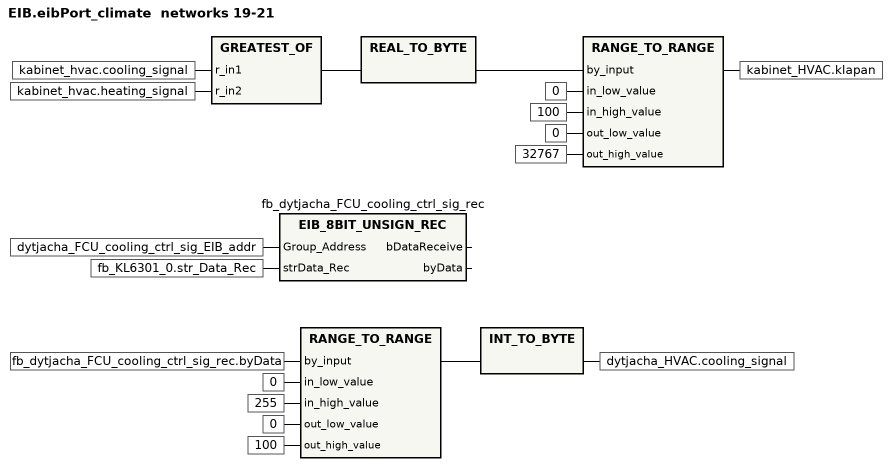
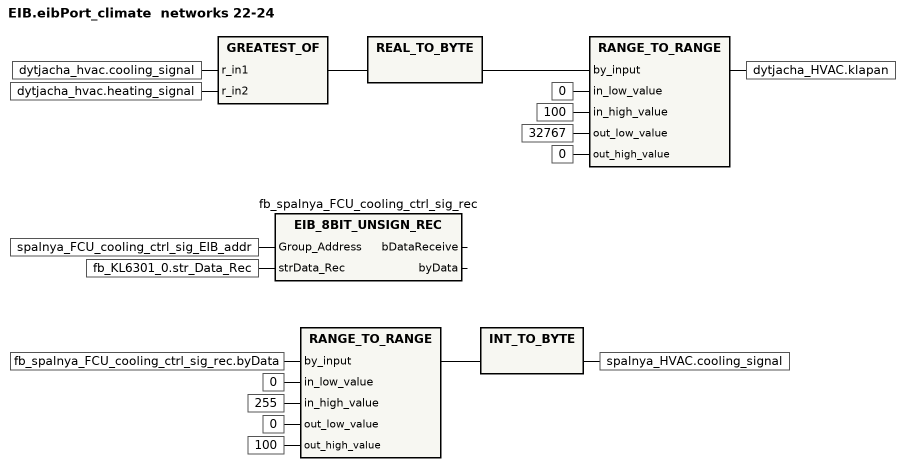
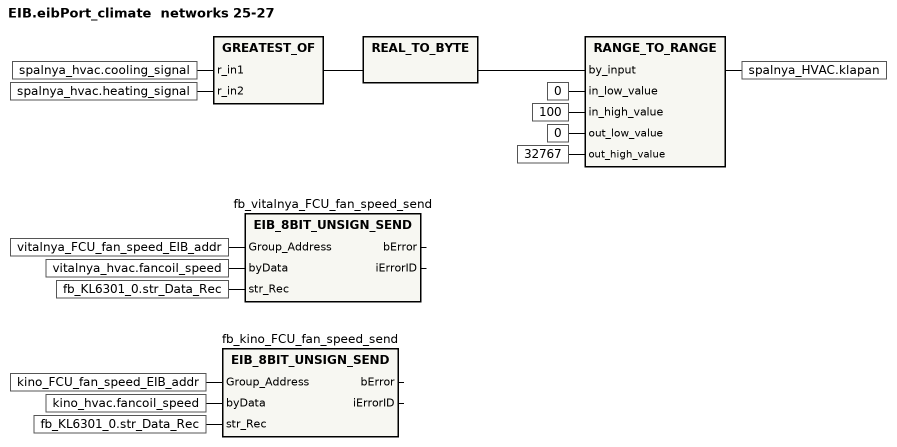
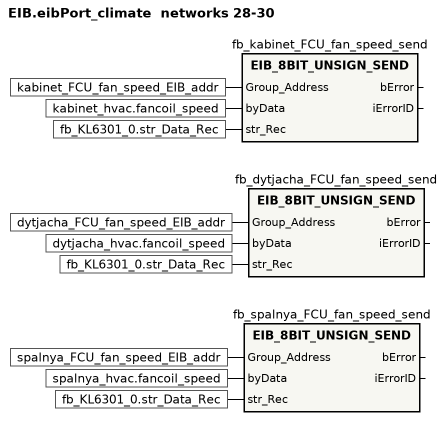
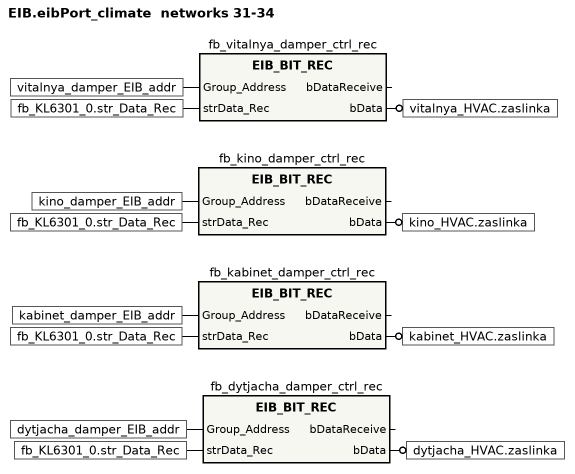
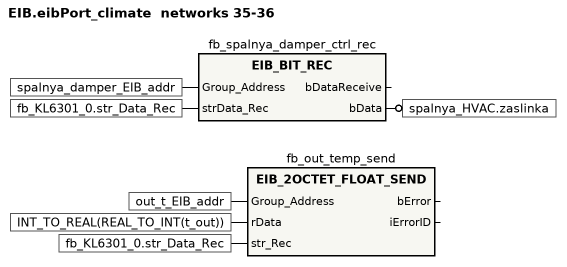
_FBD_ (* Function Block Diagram *)
NETWORK 1
	fb_vitalnya_FCU_heating_ctrl_sig_rec:EIB_8BIT_UNSIGN_REC(Group_Address: vitalnya_FCU_heating_ctrl_sig_EIB_addr, strData_Rec: fb_KL6301_0.str_Data_Rec)
NETWORK 2
	INT_TO_BYTE(RANGE_TO_RANGE(by_input: fb_vitalnya_FCU_heating_ctrl_sig_rec.byData, in_low_value: 0, in_high_value: 255, out_low_value: 0, out_high_value: 100)) => vitalnya_HVAC.heating_signal
NETWORK 3
	fb_kino_FCU_heating_ctrl_sig_rec:EIB_8BIT_UNSIGN_REC(Group_Address: kino_FCU_heating_ctrl_sig_EIB_addr, strData_Rec: fb_KL6301_0.str_Data_Rec)
NETWORK 4
	INT_TO_BYTE(RANGE_TO_RANGE(by_input: fb_kino_FCU_heating_ctrl_sig_rec.byData, in_low_value: 0, in_high_value: 255, out_low_value: 0, out_high_value: 100)) => kino_HVAC.heating_signal
NETWORK 5
	fb_kabinet_FCU_heating_ctrl_sig_rec:EIB_8BIT_UNSIGN_REC(Group_Address: kabinet_FCU_heating_ctrl_sig_EIB_addr, strData_Rec: fb_KL6301_0.str_Data_Rec)
NETWORK 6
	INT_TO_BYTE(RANGE_TO_RANGE(by_input: fb_kabinet_FCU_heating_ctrl_sig_rec.byData, in_low_value: 0, in_high_value: 255, out_low_value: 0, out_high_value: 100)) => kabinet_HVAC.heating_signal
NETWORK 7
	fb_dytjacha_FCU_heating_ctrl_sig_rec:EIB_8BIT_UNSIGN_REC(Group_Address: dytjacha_FCU_heating_ctrl_sig_EIB_addr, strData_Rec: fb_KL6301_0.str_Data_Rec)
NETWORK 8
	INT_TO_BYTE(RANGE_TO_RANGE(by_input: fb_dytjacha_FCU_heating_ctrl_sig_rec.byData, in_low_value: 0, in_high_value: 255, out_low_value: 0, out_high_value: 100)) => dytjacha_HVAC.heating_signal
NETWORK 9
	fb_spalnya_FCU_heating_ctrl_sig_rec:EIB_8BIT_UNSIGN_REC(Group_Address: spalnya_FCU_heating_ctrl_sig_EIB_addr, strData_Rec: fb_KL6301_0.str_Data_Rec)
NETWORK 10
	INT_TO_BYTE(RANGE_TO_RANGE(by_input: fb_spalnya_FCU_heating_ctrl_sig_rec.byData, in_low_value: 0, in_high_value: 255, out_low_value: 0, out_high_value: 100)) => spalnya_HVAC.heating_signal
NETWORK 11
	fb_vitalnya_FCU_cooling_ctrl_sig_rec:EIB_8BIT_UNSIGN_REC(Group_Address: vitalnya_FCU_cooling_ctrl_sig_EIB_addr, strData_Rec: fb_KL6301_0.str_Data_Rec)
NETWORK 12
	INT_TO_BYTE(RANGE_TO_RANGE(by_input: fb_vitalnya_FCU_cooling_ctrl_sig_rec.byData, in_low_value: 0, in_high_value: 255, out_low_value: 0, out_high_value: 100)) => vitalnya_HVAC.cooling_signal
NETWORK 13
	RANGE_TO_RANGE(by_input: REAL_TO_BYTE(GREATEST_OF(r_in1: vitalnya_hvac.cooling_signal, r_in2: vitalnya_hvac.heating_signal)), in_low_value: 0, in_high_value: 100, out_low_value: 0, out_high_value: 32767) => vitalnya_HVAC.klapan
NETWORK 14
	fb_kino_FCU_cooling_ctrl_sig_rec:EIB_8BIT_UNSIGN_REC(Group_Address: kino_FCU_cooling_ctrl_sig_EIB_addr, strData_Rec: fb_KL6301_0.str_Data_Rec)
NETWORK 15
	INT_TO_BYTE(RANGE_TO_RANGE(by_input: fb_kino_FCU_cooling_ctrl_sig_rec.byData, in_low_value: 0, in_high_value: 255, out_low_value: 0, out_high_value: 100)) => kino_HVAC.cooling_signal
NETWORK 16
	RANGE_TO_RANGE(by_input: REAL_TO_BYTE(GREATEST_OF(r_in1: kino_hvac.cooling_signal, r_in2: kino_hvac.heating_signal)), in_low_value: 0, in_high_value: 100, out_low_value: 0, out_high_value: 32767) => kino_HVAC.klapan
NETWORK 17
	fb_kabinet_FCU_cooling_ctrl_sig_rec:EIB_8BIT_UNSIGN_REC(Group_Address: kabinet_FCU_cooling_ctrl_sig_EIB_addr, strData_Rec: fb_KL6301_0.str_Data_Rec)
NETWORK 18
	INT_TO_BYTE(RANGE_TO_RANGE(by_input: fb_kabinet_FCU_cooling_ctrl_sig_rec.byData, in_low_value: 0, in_high_value: 255, out_low_value: 0, out_high_value: 100)) => kabinet_HVAC.cooling_signal
NETWORK 19
	RANGE_TO_RANGE(by_input: REAL_TO_BYTE(GREATEST_OF(r_in1: kabinet_hvac.cooling_signal, r_in2: kabinet_hvac.heating_signal)), in_low_value: 0, in_high_value: 100, out_low_value: 0, out_high_value: 32767) => kabinet_HVAC.klapan
NETWORK 20
	fb_dytjacha_FCU_cooling_ctrl_sig_rec:EIB_8BIT_UNSIGN_REC(Group_Address: dytjacha_FCU_cooling_ctrl_sig_EIB_addr, strData_Rec: fb_KL6301_0.str_Data_Rec)
NETWORK 21
	INT_TO_BYTE(RANGE_TO_RANGE(by_input: fb_dytjacha_FCU_cooling_ctrl_sig_rec.byData, in_low_value: 0, in_high_value: 255, out_low_value: 0, out_high_value: 100)) => dytjacha_HVAC.cooling_signal
NETWORK 22
	RANGE_TO_RANGE(by_input: REAL_TO_BYTE(GREATEST_OF(r_in1: dytjacha_hvac.cooling_signal, r_in2: dytjacha_hvac.heating_signal)), in_low_value: 0, in_high_value: 100, out_low_value: 32767, out_high_value: 0) => dytjacha_HVAC.klapan
NETWORK 23
	fb_spalnya_FCU_cooling_ctrl_sig_rec:EIB_8BIT_UNSIGN_REC(Group_Address: spalnya_FCU_cooling_ctrl_sig_EIB_addr, strData_Rec: fb_KL6301_0.str_Data_Rec)
NETWORK 24
	INT_TO_BYTE(RANGE_TO_RANGE(by_input: fb_spalnya_FCU_cooling_ctrl_sig_rec.byData, in_low_value: 0, in_high_value: 255, out_low_value: 0, out_high_value: 100)) => spalnya_HVAC.cooling_signal
NETWORK 25
	RANGE_TO_RANGE(by_input: REAL_TO_BYTE(GREATEST_OF(r_in1: spalnya_hvac.cooling_signal, r_in2: spalnya_hvac.heating_signal)), in_low_value: 0, in_high_value: 100, out_low_value: 0, out_high_value: 32767) => spalnya_HVAC.klapan
NETWORK 26
	fb_vitalnya_FCU_fan_speed_send:EIB_8BIT_UNSIGN_SEND(Group_Address: vitalnya_FCU_fan_speed_EIB_addr, byData: vitalnya_hvac.fancoil_speed, str_Rec: fb_KL6301_0.str_Data_Rec)
NETWORK 27
	fb_kino_FCU_fan_speed_send:EIB_8BIT_UNSIGN_SEND(Group_Address: kino_FCU_fan_speed_EIB_addr, byData: kino_hvac.fancoil_speed, str_Rec: fb_KL6301_0.str_Data_Rec)
NETWORK 28
	fb_kabinet_FCU_fan_speed_send:EIB_8BIT_UNSIGN_SEND(Group_Address: kabinet_FCU_fan_speed_EIB_addr, byData: kabinet_hvac.fancoil_speed, str_Rec: fb_KL6301_0.str_Data_Rec)
NETWORK 29
	fb_dytjacha_FCU_fan_speed_send:EIB_8BIT_UNSIGN_SEND(Group_Address: dytjacha_FCU_fan_speed_EIB_addr, byData: dytjacha_hvac.fancoil_speed, str_Rec: fb_KL6301_0.str_Data_Rec)
NETWORK 30
	fb_spalnya_FCU_fan_speed_send:EIB_8BIT_UNSIGN_SEND(Group_Address: spalnya_FCU_fan_speed_EIB_addr, byData: spalnya_hvac.fancoil_speed, str_Rec: fb_KL6301_0.str_Data_Rec)
NETWORK 31
	fb_vitalnya_damper_ctrl_rec:EIB_BIT_REC(Group_Address: vitalnya_damper_EIB_addr, strData_Rec: fb_KL6301_0.str_Data_Rec, bData => NOT vitalnya_HVAC.zaslinka)
NETWORK 32
	fb_kino_damper_ctrl_rec:EIB_BIT_REC(Group_Address: kino_damper_EIB_addr, strData_Rec: fb_KL6301_0.str_Data_Rec, bData => NOT kino_HVAC.zaslinka)
NETWORK 33
	fb_kabinet_damper_ctrl_rec:EIB_BIT_REC(Group_Address: kabinet_damper_EIB_addr, strData_Rec: fb_KL6301_0.str_Data_Rec, bData => NOT kabinet_HVAC.zaslinka)
NETWORK 34
	fb_dytjacha_damper_ctrl_rec:EIB_BIT_REC(Group_Address: dytjacha_damper_EIB_addr, strData_Rec: fb_KL6301_0.str_Data_Rec, bData => NOT dytjacha_HVAC.zaslinka)
NETWORK 35
	fb_spalnya_damper_ctrl_rec:EIB_BIT_REC(Group_Address: spalnya_damper_EIB_addr, strData_Rec: fb_KL6301_0.str_Data_Rec, bData => NOT spalnya_HVAC.zaslinka)
NETWORK 36
	fb_out_temp_send:EIB_2OCTET_FLOAT_SEND(Group_Address: out_t_EIB_addr, rData: INT_TO_REAL(REAL_TO_INT(t_out)), str_Rec: fb_KL6301_0.str_Data_Rec)
_END_FBD_
(* the same logic as Structured Text *)
(* Network 1 *)
fb_vitalnya_FCU_heating_ctrl_sig_rec(Group_Address := vitalnya_FCU_heating_ctrl_sig_EIB_addr, strData_Rec := fb_KL6301_0.str_Data_Rec);
(* Network 2 *)
vitalnya_HVAC.heating_signal := INT_TO_BYTE(RANGE_TO_RANGE(by_input := fb_vitalnya_FCU_heating_ctrl_sig_rec.byData, in_low_value := 0, in_high_value := 255, out_low_value := 0, out_high_value := 100));
(* Network 3 *)
fb_kino_FCU_heating_ctrl_sig_rec(Group_Address := kino_FCU_heating_ctrl_sig_EIB_addr, strData_Rec := fb_KL6301_0.str_Data_Rec);
(* Network 4 *)
kino_HVAC.heating_signal := INT_TO_BYTE(RANGE_TO_RANGE(by_input := fb_kino_FCU_heating_ctrl_sig_rec.byData, in_low_value := 0, in_high_value := 255, out_low_value := 0, out_high_value := 100));
(* Network 5 *)
fb_kabinet_FCU_heating_ctrl_sig_rec(Group_Address := kabinet_FCU_heating_ctrl_sig_EIB_addr, strData_Rec := fb_KL6301_0.str_Data_Rec);
(* Network 6 *)
kabinet_HVAC.heating_signal := INT_TO_BYTE(RANGE_TO_RANGE(by_input := fb_kabinet_FCU_heating_ctrl_sig_rec.byData, in_low_value := 0, in_high_value := 255, out_low_value := 0, out_high_value := 100));
(* Network 7 *)
fb_dytjacha_FCU_heating_ctrl_sig_rec(Group_Address := dytjacha_FCU_heating_ctrl_sig_EIB_addr, strData_Rec := fb_KL6301_0.str_Data_Rec);
(* Network 8 *)
dytjacha_HVAC.heating_signal := INT_TO_BYTE(RANGE_TO_RANGE(by_input := fb_dytjacha_FCU_heating_ctrl_sig_rec.byData, in_low_value := 0, in_high_value := 255, out_low_value := 0, out_high_value := 100));
(* Network 9 *)
fb_spalnya_FCU_heating_ctrl_sig_rec(Group_Address := spalnya_FCU_heating_ctrl_sig_EIB_addr, strData_Rec := fb_KL6301_0.str_Data_Rec);
(* Network 10 *)
spalnya_HVAC.heating_signal := INT_TO_BYTE(RANGE_TO_RANGE(by_input := fb_spalnya_FCU_heating_ctrl_sig_rec.byData, in_low_value := 0, in_high_value := 255, out_low_value := 0, out_high_value := 100));
(* Network 11 *)
fb_vitalnya_FCU_cooling_ctrl_sig_rec(Group_Address := vitalnya_FCU_cooling_ctrl_sig_EIB_addr, strData_Rec := fb_KL6301_0.str_Data_Rec);
(* Network 12 *)
vitalnya_HVAC.cooling_signal := INT_TO_BYTE(RANGE_TO_RANGE(by_input := fb_vitalnya_FCU_cooling_ctrl_sig_rec.byData, in_low_value := 0, in_high_value := 255, out_low_value := 0, out_high_value := 100));
(* Network 13 *)
vitalnya_HVAC.klapan := RANGE_TO_RANGE(by_input := REAL_TO_BYTE(GREATEST_OF(r_in1 := vitalnya_hvac.cooling_signal, r_in2 := vitalnya_hvac.heating_signal)), in_low_value := 0, in_high_value := 100, out_low_value := 0, out_high_value := 32767);
(* Network 14 *)
fb_kino_FCU_cooling_ctrl_sig_rec(Group_Address := kino_FCU_cooling_ctrl_sig_EIB_addr, strData_Rec := fb_KL6301_0.str_Data_Rec);
(* Network 15 *)
kino_HVAC.cooling_signal := INT_TO_BYTE(RANGE_TO_RANGE(by_input := fb_kino_FCU_cooling_ctrl_sig_rec.byData, in_low_value := 0, in_high_value := 255, out_low_value := 0, out_high_value := 100));
(* Network 16 *)
kino_HVAC.klapan := RANGE_TO_RANGE(by_input := REAL_TO_BYTE(GREATEST_OF(r_in1 := kino_hvac.cooling_signal, r_in2 := kino_hvac.heating_signal)), in_low_value := 0, in_high_value := 100, out_low_value := 0, out_high_value := 32767);
(* Network 17 *)
fb_kabinet_FCU_cooling_ctrl_sig_rec(Group_Address := kabinet_FCU_cooling_ctrl_sig_EIB_addr, strData_Rec := fb_KL6301_0.str_Data_Rec);
(* Network 18 *)
kabinet_HVAC.cooling_signal := INT_TO_BYTE(RANGE_TO_RANGE(by_input := fb_kabinet_FCU_cooling_ctrl_sig_rec.byData, in_low_value := 0, in_high_value := 255, out_low_value := 0, out_high_value := 100));
(* Network 19 *)
kabinet_HVAC.klapan := RANGE_TO_RANGE(by_input := REAL_TO_BYTE(GREATEST_OF(r_in1 := kabinet_hvac.cooling_signal, r_in2 := kabinet_hvac.heating_signal)), in_low_value := 0, in_high_value := 100, out_low_value := 0, out_high_value := 32767);
(* Network 20 *)
fb_dytjacha_FCU_cooling_ctrl_sig_rec(Group_Address := dytjacha_FCU_cooling_ctrl_sig_EIB_addr, strData_Rec := fb_KL6301_0.str_Data_Rec);
(* Network 21 *)
dytjacha_HVAC.cooling_signal := INT_TO_BYTE(RANGE_TO_RANGE(by_input := fb_dytjacha_FCU_cooling_ctrl_sig_rec.byData, in_low_value := 0, in_high_value := 255, out_low_value := 0, out_high_value := 100));
(* Network 22 *)
dytjacha_HVAC.klapan := RANGE_TO_RANGE(by_input := REAL_TO_BYTE(GREATEST_OF(r_in1 := dytjacha_hvac.cooling_signal, r_in2 := dytjacha_hvac.heating_signal)), in_low_value := 0, in_high_value := 100, out_low_value := 32767, out_high_value := 0);
(* Network 23 *)
fb_spalnya_FCU_cooling_ctrl_sig_rec(Group_Address := spalnya_FCU_cooling_ctrl_sig_EIB_addr, strData_Rec := fb_KL6301_0.str_Data_Rec);
(* Network 24 *)
spalnya_HVAC.cooling_signal := INT_TO_BYTE(RANGE_TO_RANGE(by_input := fb_spalnya_FCU_cooling_ctrl_sig_rec.byData, in_low_value := 0, in_high_value := 255, out_low_value := 0, out_high_value := 100));
(* Network 25 *)
spalnya_HVAC.klapan := RANGE_TO_RANGE(by_input := REAL_TO_BYTE(GREATEST_OF(r_in1 := spalnya_hvac.cooling_signal, r_in2 := spalnya_hvac.heating_signal)), in_low_value := 0, in_high_value := 100, out_low_value := 0, out_high_value := 32767);
(* Network 26 *)
fb_vitalnya_FCU_fan_speed_send(Group_Address := vitalnya_FCU_fan_speed_EIB_addr, byData := vitalnya_hvac.fancoil_speed, str_Rec := fb_KL6301_0.str_Data_Rec);
(* Network 27 *)
fb_kino_FCU_fan_speed_send(Group_Address := kino_FCU_fan_speed_EIB_addr, byData := kino_hvac.fancoil_speed, str_Rec := fb_KL6301_0.str_Data_Rec);
(* Network 28 *)
fb_kabinet_FCU_fan_speed_send(Group_Address := kabinet_FCU_fan_speed_EIB_addr, byData := kabinet_hvac.fancoil_speed, str_Rec := fb_KL6301_0.str_Data_Rec);
(* Network 29 *)
fb_dytjacha_FCU_fan_speed_send(Group_Address := dytjacha_FCU_fan_speed_EIB_addr, byData := dytjacha_hvac.fancoil_speed, str_Rec := fb_KL6301_0.str_Data_Rec);
(* Network 30 *)
fb_spalnya_FCU_fan_speed_send(Group_Address := spalnya_FCU_fan_speed_EIB_addr, byData := spalnya_hvac.fancoil_speed, str_Rec := fb_KL6301_0.str_Data_Rec);
(* Network 31 *)
fb_vitalnya_damper_ctrl_rec(Group_Address := vitalnya_damper_EIB_addr, strData_Rec := fb_KL6301_0.str_Data_Rec);
vitalnya_HVAC.zaslinka := NOT fb_vitalnya_damper_ctrl_rec.bData;
(* Network 32 *)
fb_kino_damper_ctrl_rec(Group_Address := kino_damper_EIB_addr, strData_Rec := fb_KL6301_0.str_Data_Rec);
kino_HVAC.zaslinka := NOT fb_kino_damper_ctrl_rec.bData;
(* Network 33 *)
fb_kabinet_damper_ctrl_rec(Group_Address := kabinet_damper_EIB_addr, strData_Rec := fb_KL6301_0.str_Data_Rec);
kabinet_HVAC.zaslinka := NOT fb_kabinet_damper_ctrl_rec.bData;
(* Network 34 *)
fb_dytjacha_damper_ctrl_rec(Group_Address := dytjacha_damper_EIB_addr, strData_Rec := fb_KL6301_0.str_Data_Rec);
dytjacha_HVAC.zaslinka := NOT fb_dytjacha_damper_ctrl_rec.bData;
(* Network 35 *)
fb_spalnya_damper_ctrl_rec(Group_Address := spalnya_damper_EIB_addr, strData_Rec := fb_KL6301_0.str_Data_Rec);
spalnya_HVAC.zaslinka := NOT fb_spalnya_damper_ctrl_rec.bData;
(* Network 36 *)
fb_out_temp_send(Group_Address := out_t_EIB_addr, rData := INT_TO_REAL(REAL_TO_INT(t_out)), str_Rec := fb_KL6301_0.str_Data_Rec);
END_ACTION
ACTION floor1:
data1floor[0].5:=bDarkOutside;
data1floor[0].6:=Light.tambur3_2_short_click;
data1floor[0].7:=Light.tambur3_2_long_click;

data1floor[4]:=WORD_TO_BYTE(system_time.wHour);
data1floor[5]:=WORD_TO_BYTE(system_time.wMinute);

MEMCPY(ADR(data1floor[10] ), ADR(OAT), SIZEOF(OAT));

fb_komora_l_read(strData_Rec:=fb_KL6301_0.str_Data_Rec,   Group_Address:=komora_l_adr);
IF NOT  fb_komora_l_read.bDataReceive THEN
	data1floor[100].0:= fb_komora_l_read.bdata;
END_IF

fb_su1_l_read(strData_Rec:=fb_KL6301_0.str_Data_Rec,   Group_Address:=su1_l_adr);
IF NOT  fb_su1_l_read.bDataReceive THEN
	data1floor[100].1:= fb_su1_l_read.bdata;
END_IF

fb_topochna_l_read(strData_Rec:=fb_KL6301_0.str_Data_Rec,  Group_Address:=topochna_l_adr);
IF NOT  fb_topochna_l_read.bDataReceive THEN
	data1floor[100].2:= fb_topochna_l_read.bdata;
END_IF

fb_su2_bra_read(strData_Rec:=fb_KL6301_0.str_Data_Rec, Group_Address:=su2_bra_adr);
IF NOT  fb_su2_bra_read.bDataReceive THEN
	data1floor[100].3:= fb_su2_bra_read.bdata;
END_IF

fb_su2_l_read(strData_Rec:=fb_KL6301_0.str_Data_Rec, Group_Address:=su2_l_adr);
IF NOT  fb_su2_l_read.bDataReceive THEN
	data1floor[100].4:= fb_su2_l_read.bdata;
END_IF

fb_su1_rakovyna_read(strData_Rec:=fb_KL6301_0.str_Data_Rec, Group_Address:=su1_rakovyna_adr);
IF NOT  fb_su1_rakovyna_read.bDataReceive THEN
	data1floor[100].5:= fb_su1_rakovyna_read.bdata;
END_IF

fb_su2_dush_read(strData_Rec:=fb_KL6301_0.str_Data_Rec, Group_Address:=su2_dush_adr);
IF NOT  fb_su2_dush_read.bDataReceive THEN
	data1floor[100].6:= fb_su2_dush_read.bdata;
END_IF

fb_dush_read(strData_Rec:=fb_KL6301_0.str_Data_Rec, Group_Address:=dush_adr);
IF NOT  fb_dush_read.bDataReceive THEN
	data1floor[100].7:= fb_dush_read.bdata;
END_IF

fb_kuhnya1_read(strData_Rec:=fb_KL6301_0.str_Data_Rec, Group_Address:=kuhnya1_adr);
IF NOT  fb_kuhnya1_read.bDataReceive THEN
	data1floor[101].0:= fb_kuhnya1_read.bdata;
END_IF

fb_vitalnya_smugy1_read(strData_Rec:=fb_KL6301_0.str_Data_Rec, Group_Address:=vitalnya_smugy1_adr);
IF NOT  fb_vitalnya_smugy1_read.bDataReceive THEN
	data1floor[101].1:= fb_vitalnya_smugy1_read.bdata;
END_IF

fb_vitalnya_l_read(strData_Rec:=fb_KL6301_0.str_Data_Rec, Group_Address:=vitalnya_l_adr);
IF NOT  fb_vitalnya_l_read.bDataReceive THEN
	data1floor[101].2:= fb_vitalnya_l_read.bdata;
END_IF

fb_vitalnya_prokladka_read(strData_Rec:=fb_KL6301_0.str_Data_Rec, Group_Address:=vitalnya_prokladka_adr);
IF NOT  fb_vitalnya_prokladka_read.bDataReceive THEN
	data1floor[101].3:= fb_vitalnya_prokladka_read.bdata;
END_IF

fb_terassa_stina_read(strData_Rec:=fb_KL6301_0.str_Data_Rec, Group_Address:=terassa_stina_adr);
IF NOT  fb_terassa_stina_read.bDataReceive THEN
	data1floor[101].4:= fb_terassa_stina_read.bdata;
END_IF

fb_pidval_shody_read(strData_Rec:=fb_KL6301_0.str_Data_Rec, Group_Address:=pidval_shody_adr);
IF NOT  fb_pidval_shody_read.bDataReceive THEN
	data1floor[101].5:= fb_pidval_shody_read.bdata;
END_IF

fb_skhody2pov_read(strData_Rec:=fb_KL6301_0.str_Data_Rec, Group_Address:=skhody2pov_adr);
IF NOT  fb_skhody2pov_read.bDataReceive THEN
	data1floor[101].6:= fb_skhody2pov_read.bdata;
END_IF

fb_tambur_l_read(strData_Rec:=fb_KL6301_0.str_Data_Rec, Group_Address:=tambur_l_adr);
IF NOT  fb_tambur_l_read.bDataReceive THEN
	data1floor[101].7:= fb_tambur_l_read.bdata;
END_IF

fb_vent_su1_read(strData_Rec:=fb_KL6301_0.str_Data_Rec, Group_Address:=vent_su1_adr);
IF NOT  fb_vent_su1_read.bDataReceive THEN
	data1floor[102].0:= fb_vent_su1_read.bdata;
END_IF

fb_vent_kuh_low_read(strData_Rec:=fb_KL6301_0.str_Data_Rec, Group_Address:=vent_kuh_low_adr);
IF NOT  fb_vent_kuh_low_read.bDataReceive THEN
	data1floor[102].1:= fb_vent_kuh_low_read.bdata;
END_IF

fb_vent_dush_read(strData_Rec:=fb_KL6301_0.str_Data_Rec, Group_Address:=vent_dush_adr);
IF NOT  fb_vent_dush_read.bDataReceive THEN
	data1floor[102].2:= fb_vent_dush_read.bdata;
END_IF

fb_vent_komora_read(strData_Rec:=fb_KL6301_0.str_Data_Rec, Group_Address:=vent_komora_adr);
IF NOT  fb_vent_komora_read.bDataReceive THEN
	data1floor[102].3:= fb_vent_komora_read.bdata;
END_IF

fb_vent_kuh_high_read(strData_Rec:=fb_KL6301_0.str_Data_Rec, Group_Address:=vent_kuh_high_adr);
IF NOT  fb_vent_kuh_high_read.bDataReceive THEN
	data1floor[102].4:= fb_vent_kuh_high_read.bdata;
END_IF

(*sending*)
fb_komora_l_send_status_ex(imode:=eib_send_mode_floor1, bStart:=eib_send_cyclical_start_floor1, str_Rec:=fb_KL6301_0.str_Data_Rec, bData:=komora_l,  Group_Address:=komora_l_status_adr);
fb_su1_l_send_status_ex(imode:=eib_send_mode_floor1, bStart:=eib_send_cyclical_start_floor1, str_Rec:=fb_KL6301_0.str_Data_Rec, bData:=su1_l,  Group_Address:=su1_l_status_adr);
fb_topochna_l_send_status_ex(imode:=eib_send_mode_floor1, bStart:=eib_send_cyclical_start_floor1, str_Rec:=fb_KL6301_0.str_Data_Rec, bData:=topochna_l,  Group_Address:=topochna_l_status_adr);
fb_su2_bra_send_status_ex(imode:=eib_send_mode_floor1, bStart:=eib_send_cyclical_start_floor1, str_Rec:=fb_KL6301_0.str_Data_Rec, bData:=su2_bra,  Group_Address:=su2_bra_status_adr);
fb_su2_l_send_status_ex(imode:=eib_send_mode_floor1, bStart:=eib_send_cyclical_start_floor1, str_Rec:=fb_KL6301_0.str_Data_Rec, bData:=su2_l,  Group_Address:=su2_l_status_adr);
fb_su1_rakovyna_send_status_ex(imode:=eib_send_mode_floor1, bStart:=eib_send_cyclical_start_floor1, str_Rec:=fb_KL6301_0.str_Data_Rec, bData:=su1_rakovyna,  Group_Address:=su1_rakovyna_status_adr);
fb_su2_dush_send_status_ex(imode:=eib_send_mode_floor1, bStart:=eib_send_cyclical_start_floor1, str_Rec:=fb_KL6301_0.str_Data_Rec, bData:=su2_dush,  Group_Address:=su2_dush_status_adr);
fb_dush_send_status_ex(imode:=eib_send_mode_floor1, bStart:=eib_send_cyclical_start_floor1, str_Rec:=fb_KL6301_0.str_Data_Rec, bData:=dush,  Group_Address:=dush_status_adr);
fb_kuhnya1_send_status_ex(imode:=eib_send_mode_floor1, bStart:=eib_send_cyclical_start_floor1, str_Rec:=fb_KL6301_0.str_Data_Rec, bData:=kuhnya1,  Group_Address:=kuhnya1_status_adr);
fb_vitalnya_smugy1_send_status_ex(imode:=eib_send_mode_floor1, bStart:=eib_send_cyclical_start_floor1, str_Rec:=fb_KL6301_0.str_Data_Rec, bData:=vitalnya_smugy1,  Group_Address:=vitalnya_smugy1_status_adr);
fb_vitalnya_l_send_status_ex(imode:=eib_send_mode_floor1, bStart:=eib_send_cyclical_start_floor1, str_Rec:=fb_KL6301_0.str_Data_Rec, bData:=vitalnya_l,  Group_Address:=vitalnya_l_status_adr);
fb_vitalnya_prokladka_send_status_ex(imode:=eib_send_mode_floor1, bStart:=eib_send_cyclical_start_floor1, str_Rec:=fb_KL6301_0.str_Data_Rec, bData:=vitalnya_prokladka,  Group_Address:=vitalnya_prokladka_status_adr);
fb_terassa_stina_send_status_ex(imode:=eib_send_mode_floor1, bStart:=eib_send_cyclical_start_floor1, str_Rec:=fb_KL6301_0.str_Data_Rec, bData:=terassa_stina,  Group_Address:=terassa_stina_status_adr);
fb_pidval_shody_send_status_ex(imode:=eib_send_mode_floor1, bStart:=eib_send_cyclical_start_floor1, str_Rec:=fb_KL6301_0.str_Data_Rec, bData:=pidval_shody,  Group_Address:=pidval_shody_status_adr);
fb_skhody2pov_send_status_ex(imode:=eib_send_mode_floor1, bStart:=eib_send_cyclical_start_floor1, str_Rec:=fb_KL6301_0.str_Data_Rec, bData:=skhody2pov,  Group_Address:=skhody2pov_status_adr);
fb_tambur_l_send_status_ex(imode:=eib_send_mode_floor1, bStart:=eib_send_cyclical_start_floor1, str_Rec:=fb_KL6301_0.str_Data_Rec, bData:=tambur_l,  Group_Address:=tambur_l_status_adr);
fb_vent_su1_send_status_ex(imode:=eib_send_mode_floor1, bStart:=eib_send_cyclical_start_floor1, str_Rec:=fb_KL6301_0.str_Data_Rec, bData:=vent_su1,  Group_Address:=vent_su1_status_adr);
fb_vent_kuh_low_send_status_ex(imode:=eib_send_mode_floor1, bStart:=eib_send_cyclical_start_floor1, str_Rec:=fb_KL6301_0.str_Data_Rec, bData:=vent_kuh_low,  Group_Address:=vent_kuh_low_status_adr);
fb_vent_dush_send_status_ex(imode:=eib_send_mode_floor1, bStart:=eib_send_cyclical_start_floor1, str_Rec:=fb_KL6301_0.str_Data_Rec, bData:=vent_dush,  Group_Address:=vent_dush_status_adr);
fb_vent_komora_send_status_ex(imode:=eib_send_mode_floor1, bStart:=eib_send_cyclical_start_floor1, str_Rec:=fb_KL6301_0.str_Data_Rec, bData:=vent_komora,  Group_Address:=vent_komora_status_adr);
fb_vent_kuh_high_send_status_ex(imode:=eib_send_mode_floor1, bStart:=eib_send_cyclical_start_floor1, str_Rec:=fb_KL6301_0.str_Data_Rec, bData:=vent_kuh_high,  Group_Address:=vent_kuh_high_status_adr);

IF fb_komora_l_send_status_ex.bBusy OR fb_heartbeat_timer.Q   THEN
	data1floor[100].0:=komora_l;
END_IF

IF fb_su1_l_send_status_ex.bBusy OR fb_heartbeat_timer.Q   THEN
	data1floor[100].1:=su1_l;
END_IF

IF fb_topochna_l_send_status_ex.bBusy OR fb_heartbeat_timer.Q   THEN
	data1floor[100].2:=topochna_l;
END_IF

IF fb_su2_bra_send_status_ex.bBusy OR fb_heartbeat_timer.Q   THEN
	data1floor[100].3:=su2_bra;
END_IF

IF fb_su2_l_send_status_ex.bBusy OR fb_heartbeat_timer.Q   THEN
	data1floor[100].4:=su2_l;
END_IF

IF fb_su1_rakovyna_send_status_ex.bBusy OR fb_heartbeat_timer.Q   THEN
	data1floor[100].5:=su1_rakovyna;
END_IF

IF fb_su2_dush_send_status_ex.bBusy OR fb_heartbeat_timer.Q   THEN
	data1floor[100].6:=su2_dush;
END_IF

IF fb_dush_send_status_ex.bBusy OR fb_heartbeat_timer.Q   THEN
	data1floor[100].7:=dush;
END_IF

IF fb_kuhnya1_send_status_ex.bBusy OR fb_heartbeat_timer.Q  THEN
	data1floor[101].0:=kuhnya1;
END_IF

IF fb_vitalnya_smugy1_send_status_ex.bBusy OR fb_heartbeat_timer.Q   THEN
	data1floor[101].1:=vitalnya_smugy1;
END_IF

IF fb_vitalnya_l_send_status_ex.bBusy OR fb_heartbeat_timer.Q   THEN
	data1floor[101].2:=vitalnya_l;
END_IF

IF fb_vitalnya_prokladka_send_status_ex.bBusy OR fb_heartbeat_timer.Q   THEN
	data1floor[101].3:=vitalnya_prokladka;
END_IF

IF fb_terassa_stina_send_status_ex.bBusy OR fb_heartbeat_timer.Q   THEN
	data1floor[101].4:=terassa_stina;
END_IF

IF fb_pidval_shody_send_status_ex.bBusy OR fb_heartbeat_timer.Q   THEN
	data1floor[101].5:=pidval_shody;
END_IF

IF fb_skhody2pov_send_status_ex.bBusy OR fb_heartbeat_timer.Q   THEN
	data1floor[101].6:=skhody2pov;
END_IF

IF fb_tambur_l_send_status_ex.bBusy OR fb_heartbeat_timer.Q   THEN
	data1floor[101].7:=tambur_l;
END_IF

IF fb_vent_su1_send_status_ex.bBusy OR fb_heartbeat_timer.Q   THEN
	data1floor[102].0:=vent_su1;
END_IF

IF fb_vent_kuh_low_send_status_ex.bBusy OR fb_heartbeat_timer.Q   THEN
	data1floor[102].1:=vent_kuh_low;
END_IF

IF fb_vent_dush_send_status_ex.bBusy OR fb_heartbeat_timer.Q   THEN
	data1floor[102].2:=vent_dush;
END_IF

IF fb_vent_komora_send_status_ex.bBusy OR fb_heartbeat_timer.Q   THEN
	data1floor[102].3:=vent_komora;
END_IF

IF fb_vent_kuh_high_send_status_ex.bBusy OR fb_heartbeat_timer.Q   THEN
	data1floor[102].4:=vent_kuh_high;
END_IF
END_ACTION
ACTION floor2:
data2floor[6].0:=Light.tambur3_2_short_click;
data2floor[6].1:=bDarkOutside;
data2floor[6].2:=Light.tambur3_2_long_click;


data2floor[9]:=WORD_TO_BYTE(system_time.wHour);
data2floor[10]:=WORD_TO_BYTE(system_time.wMinute);

MEMCPY(ADR(data2floor[22] ), ADR(OAT), SIZEOF(OAT));

MEMCPY(ADR(KABINET_HVAC.floor_T), ADR(kabinet_floor_T_byte0), 4);
MEMCPY(ADR(STUDIO_HVAC.floor_T), ADR(studio_floor_T_byte0),  4);

fb_balkon_peryla_read(strData_Rec:=fb_KL6301_0.str_Data_Rec,   Group_Address:=balkon_peryla_adr);
IF NOT  fb_balkon_peryla_read.bDataReceive OR NOT fb_eib_twillight_rec.bDataReceive  THEN
	data2floor[100].0:= fb_balkon_peryla_read.bdata OR  fb_eib_twillight_rec.bData ;
END_IF
fb_kino_l_read(strData_Rec:=fb_KL6301_0.str_Data_Rec,   Group_Address:=kino_l_adr);
IF NOT  fb_kino_l_read.bDataReceive THEN
	data2floor[100].1:= fb_kino_l_read.bdata;
END_IF
fb_balkon_bra_read(strData_Rec:=fb_KL6301_0.str_Data_Rec,   Group_Address:=balkon_bra_adr);
IF NOT  fb_balkon_bra_read.bDataReceive OR NOT fb_eib_twillight_rec.bDataReceive THEN
	data2floor[100].2:= fb_balkon_bra_read.bdata OR fb_eib_twillight_rec.bData;
END_IF
fb_kabinet_balkon_l_read(strData_Rec:=fb_KL6301_0.str_Data_Rec,   Group_Address:=kabinet_balkon_l_adr);
IF NOT  fb_kabinet_balkon_l_read.bDataReceive THEN
	data2floor[100].3:= fb_kabinet_balkon_l_read.bdata;
END_IF
fb_balkon_read(strData_Rec:=fb_KL6301_0.str_Data_Rec,   Group_Address:=balkon_adr);
IF NOT  fb_balkon_read.bDataReceive THEN
	data2floor[100].4:= fb_balkon_read.bdata;
END_IF
fb_korydor1_read(strData_Rec:=fb_KL6301_0.str_Data_Rec,   Group_Address:=korydor1_adr);
IF NOT  fb_korydor1_read.bDataReceive THEN
	data2floor[100].5:= fb_korydor1_read.bdata;
END_IF
fb_kino_bra_read(strData_Rec:=fb_KL6301_0.str_Data_Rec,   Group_Address:=kino_bra_adr);
IF NOT  fb_kino_bra_read.bDataReceive THEN
	data2floor[100].6:= fb_kino_bra_read.bdata;
END_IF
fb_studio_pidsvitka_read(strData_Rec:=fb_KL6301_0.str_Data_Rec,   Group_Address:=studio_pidsvitka_adr);
IF NOT  fb_studio_pidsvitka_read.bDataReceive THEN
	data2floor[100].7:= fb_studio_pidsvitka_read.bdata;
END_IF
fb_skhody2_3_read(strData_Rec:=fb_KL6301_0.str_Data_Rec,   Group_Address:=skhody2_3_adr);
IF NOT  fb_skhody2_3_read.bDataReceive THEN
	data2floor[101].0:= fb_skhody2_3_read.bdata;
END_IF
fb_studio_l_read(strData_Rec:=fb_KL6301_0.str_Data_Rec,   Group_Address:=studio_l_adr);
IF NOT  fb_studio_l_read.bDataReceive THEN
	data2floor[101].1:= fb_studio_l_read.bdata;
END_IF
fb_kabinet_svitlo_read(strData_Rec:=fb_KL6301_0.str_Data_Rec,   Group_Address:=kabinet_svitlo_adr);
IF NOT  fb_kabinet_svitlo_read.bDataReceive THEN
	data2floor[101].2:= fb_kabinet_svitlo_read.bdata;
END_IF
fb_kabinet_kobra_read(strData_Rec:=fb_KL6301_0.str_Data_Rec,   Group_Address:=kabinet_kobra_adr);
IF NOT  fb_kabinet_kobra_read.bDataReceive THEN
	data2floor[101].3:= fb_kabinet_kobra_read.bdata;
END_IF
fb_tambur2_read(strData_Rec:=fb_KL6301_0.str_Data_Rec,   Group_Address:=tambur2_adr);
IF NOT  fb_tambur2_read.bDataReceive THEN
	data2floor[101].4:= fb_tambur2_read.bdata;
END_IF
fb_stend_read(strData_Rec:=fb_KL6301_0.str_Data_Rec,   Group_Address:=stend_adr);
IF NOT  fb_stend_read.bDataReceive THEN
	data2floor[101].5:= fb_stend_read.bdata;
END_IF
fb_skhody_peryla_read(strData_Rec:=fb_KL6301_0.str_Data_Rec,   Group_Address:=skhody_peryla_adr);
IF NOT  fb_skhody_peryla_read.bDataReceive OR NOT  fb_eib_twillight_rec.bDataReceive THEN
	data2floor[101].6:= fb_skhody_peryla_read.bdata OR  fb_eib_twillight_rec.bData;
END_IF

fb_kino_bra_dim_read(strData_Rec:=fb_KL6301_0.str_Data_Rec,   Group_Address:=kino_bra_dimming_adr);
IF NOT  fb_kino_bra_dim_read.bDataReceive THEN
	data2floor[102]:= INT_TO_BYTE(fb_kino_bra_dim_read.iData);
END_IF


(*sending*)
fb_balkon_peryla_send_status_ex(imode:=eib_send_mode_floor2, bStart:=eib_send_cyclical_start_floor2, str_Rec:=fb_KL6301_0.str_Data_Rec, bData:=balkon_peryla,  Group_Address:=balkon_peryla_status_adr);
fb_kino_l_send_status_ex(imode:=eib_send_mode_floor2, bStart:=eib_send_cyclical_start_floor2, str_Rec:=fb_KL6301_0.str_Data_Rec, bData:=kino_l,  Group_Address:=kino_l_status_adr);
fb_balkon_bra_send_status_ex(imode:=eib_send_mode_floor2, bStart:=eib_send_cyclical_start_floor2, str_Rec:=fb_KL6301_0.str_Data_Rec, bData:=balkon_bra,  Group_Address:=balkon_bra_status_adr);
fb_kabinet_balkon_l_send_status_ex(imode:=eib_send_mode_floor2, bStart:=eib_send_cyclical_start_floor2, str_Rec:=fb_KL6301_0.str_Data_Rec, bData:=kabinet_balkon_l,  Group_Address:=kabinet_balkon_l_status_adr);
fb_balkon_send_status_ex(imode:=eib_send_mode_floor2, bStart:=eib_send_cyclical_start_floor2, str_Rec:=fb_KL6301_0.str_Data_Rec, bData:=balkon,  Group_Address:=balkon_status_adr);
fb_korydor1_send_status_ex(imode:=eib_send_mode_floor2, bStart:=eib_send_cyclical_start_floor2, str_Rec:=fb_KL6301_0.str_Data_Rec, bData:=korydor1,  Group_Address:=korydor1_status_adr);
fb_kino_bra_send_status_ex(imode:=eib_send_mode_floor2, bStart:=eib_send_cyclical_start_floor2, str_Rec:=fb_KL6301_0.str_Data_Rec, bData:=kino_bra,  Group_Address:=kino_bra_status_adr);
fb_studio_pidsvitka_send_status_ex(imode:=eib_send_mode_floor2, bStart:=eib_send_cyclical_start_floor2, str_Rec:=fb_KL6301_0.str_Data_Rec, bData:=studio_pidsvitka,  Group_Address:=studio_pidsvitka_status_adr);
fb_skhody2_3_send_status_ex(imode:=eib_send_mode_floor2, bStart:=eib_send_cyclical_start_floor2, str_Rec:=fb_KL6301_0.str_Data_Rec, bData:=skhody2_3,  Group_Address:=skhody2_3_status_adr);
fb_studio_l_send_status_ex(imode:=eib_send_mode_floor2, bStart:=eib_send_cyclical_start_floor2, str_Rec:=fb_KL6301_0.str_Data_Rec, bData:=studio_l,  Group_Address:=studio_l_status_adr);
fb_kabinet_svitlo_send_status_ex(imode:=eib_send_mode_floor2, bStart:=eib_send_cyclical_start_floor2, str_Rec:=fb_KL6301_0.str_Data_Rec, bData:=kabinet_svitlo,  Group_Address:=kabinet_svitlo_status_adr);
fb_kabinet_kobra_send_status_ex(imode:=eib_send_mode_floor2, bStart:=eib_send_cyclical_start_floor2, str_Rec:=fb_KL6301_0.str_Data_Rec, bData:=kabinet_kobra,  Group_Address:=kabinet_kobra_status_adr);
fb_tambur2_send_status_ex(imode:=eib_send_mode_floor2, bStart:=eib_send_cyclical_start_floor2, str_Rec:=fb_KL6301_0.str_Data_Rec, bData:=tambur2,  Group_Address:=tambur2_status_adr);
fb_stend_send_status_ex(imode:=eib_send_mode_floor2, bStart:=eib_send_cyclical_start_floor2, str_Rec:=fb_KL6301_0.str_Data_Rec, bData:=stend,  Group_Address:=stend_status_adr);
fb_skhody_peryla_send_status_ex(imode:=eib_send_mode_floor2, bStart:=eib_send_cyclical_start_floor2, str_Rec:=fb_KL6301_0.str_Data_Rec, bData:=skhody_peryla,  Group_Address:=skhody_peryla_status_adr);
fb_kino_bra_send_dim_status_ex(imode:=eib_send_mode_floor2, bstart:=eib_send_cyclical_start_floor2, str_Rec:=fb_KL6301_0.str_Data_Rec, idata:=BYTE_TO_INT(kino_bra_dim_value) );

